END_VAR
VAR_OUTPUT
	stDataXelectrix					: ST_Xelectrix_Powerbox_OutData;				//Shows the specific output data from the Xelectric device
	stDataBatt						: ST_Battery_Output;							//{#lynus.ag#()} //Output structure with Data from Battery
	stDataBattInverter				: ST_BatteryInverter_Output;					//{#lynus.ag#()} //Output structure with Data from Battery Inverter
	stDataEMPower_Grid				: ST_ElectricMeter_Output_Power;				//Output structure with Data from Electric Meter Grid (Power Data)
	stDataEMCounter_Grid			: ST_ElectricMeter_Output_Counter;				//Output structure with Data from Electric Meter Grid (Counter Data)
	diNrOfBatt_OUT					: DINT;											//Active Number from the Battery Function for using on other functions
	diNrOfBattInverter_OUT			: DINT;											//Active Number from the Battery Inverter Function for using on other functions
	diNrOfEM_OUT_Grid				: DINT;											//Active Number from the Electric Meter for using on other functions
	lrMaxCapacityBattery_OUT		: LREAL;										//Max kWh from the Battery system. The Xelectrix System deliver this value.
	iSetpointPower_Info				: INT;											// Battery Setpoint, for monitoring purpose
END_VAR
VAR

	fbBattery						: FB_Battery;									//Function block for battery

	fbBatteryInverter				: FB_BatteryInverter;							//Function block for battery inveter

	fbEMGrid						: FB_ElectricMeter;								//Electric Meter Function 

	fbPIDChrgStandby				: FB_PID;										//Controller to control the battery current on 0 in the standby mode	

	fbNumberDeviceBattery			: FB_NumberOfDevice;							//Function block to calcualte the number of the Device

	fbNumberDeviceBatteryInvert		: FB_NumberOfDevice;							//Function block to calcualte the number of the Device

	fbNumberDeviceGrid				: FB_NumberOfDevice;							//Function block to calcualte the number of the Device

	fbMBRead_FC3					: FB_MBReadRegs;								//Modbus Read Function (FC3)

	fbMBWrite_FC16					: FB_MBWriteRegs;								//Modbus Write Function (FC16)

	fbConvertData					: FB_CV_WORD_TO_DWORD;							//Convert 2 Words in a Dword

	timDelay						: TON;											//Timer for Delay between Requests

	timTimeout						: TON;											//Timer for Timeout

	timDissableFunctions			: TON;											//Timer to dissable the Function after Lynus_Standards.Constants_General.tTimeDissableLynusFunctions Days without connection to the Lynus Cloud

	timResetConnectionOnGVL			: TON;											//Timer to try reset the connection Flag on the GVL. (When somebody delete the Connection Function and make only a onlinechange)

	timReset						: TON;											//Timer to reset the Inverter after a Error

	timErrorMTCP					: TON;											//Delay when Error on Modbus TCP

	timSetStandbyCntrl				: TOF;											//Timer to set the Standby Controller

	FPEnable						: R_TRIG;										//Internal positive Edge

	FPError_FC_3					: R_TRIG;										//Internal positive Edge

	FPError_FC_16					: R_TRIG;										//Internal positive Edge

	FPActivateControl				: R_TRIG;										//Internal positive Edge

	FNTimDissable					: F_TRIG;										//Internal negative Edge

	PD_String						: FB_PersistentData_String;						//Function to save persistent data

	arrPD							: ARRAY[1..7] OF FB_PersistentData_Number;		//Function to save persistent data

	arrBuffer_FC3					: ARRAY[1..48] OF WORD;							//Buffer with Data from FC3

	arrBuffer_FC16					: ARRAY[1..2] OF WORD;							//Buffer with Data from FC16

	arrCounterForGVL				: ARRAY[1..3] OF DINT;							//Counter to clean old data on GVL

	bEnergyGridConsReceived			: BOOL;											//Energy Consumption from Grid first time received

	bEnergyGridProdReceived			: BOOL;											//Energy Production from Grid first time received

	byWaitInStep					: BYTE;											//Wait in Step before start to clean data on PLC

	byLPWorkAroundACDevice			: BYTE;											//Loop for Workaround

	byNumberOfZero					: BYTE;											//Number with 0 Value from AC Messurement

	iSetpointPower					: INT;											//Power Setpoint in W

	iStateGVLData					: INT;											//State machine to handle the data on the GVL

	iStateModbusRead				: INT;											//State variable for Statemachine

	iStateModbusWrite				: INT;											//State variable for Statemachine

	iStateModbusError				: INT;											//State variable for Statemachine

	iStateModbus_CP					: INT;											//Compare State variable

	iMaxDcDischargeCurrentBattery	: INT;											//Variable to convert from negative to positive value

	diLPForGVL						: DINT;											//Loop to clean old data on GVL

	lrEnergyGridConsumption_CP		: LREAL;										//Energy Consumption from Grid for calculation for Workaround why Xelectrix send sometimes big value 

	lrEnergyGridProduction_CP		: LREAL;										//Energy Production from Grid for calculation for Workaround why Xelectrix send sometimes big value 
END_VAR
VAR PERSISTENT
	{attribute 'conditionalshow'}
	diNrOfEMS_IN_CP					: DINT;											//Number of EMS what control this Device to compare with the original
END_VAR

//Creator : Stefan Lackner (based on Kai Ebensperger V1)
//Company : EfficientIO
//Date : 15.12.2022
//Version : 2.0.0.0

//With this function its possible to read out values from the Xelectrix Powerbox from the factory Xelectrix
//Its also possible to controll the power in and out from Battery if its necessary.
//The protocol to the Inverter/powerbox is Modbus TCP
//When this Function is not enabled, then the Inverter is not off. But no power flows into or out of the battery.
//This Inverter deliver also the Grid power (smart Meter).
//Versions that are supported : 106
//NOTE : This Function block not support the complete emergency power mode. He switch not off when the byMaxDepthOfDischargeEPO is reached because this make the inverter by himself.

//NOTE for diNr.....Designation => 
//_IN = Here Data come in from other Functions or go out to other functions about the GVL
//_OUT = Here Data go out to other functions about the GVL

(*------------------------------------------------------------------------------------------General Input Part---------------------------------------------------------------------------------------------*)

//Check limitation
diNrOfEMS_IN := LIMIT(0,diNrOfEMS_IN,Constants_Energy.diMaxNumberOfEMS);
	
(*-------------------------------------------------------------Calcualte the number of Battery system---------------------------------------------------------------*)

fbNumberDeviceBattery(
	diActualNumberOfDevices:= Lynus_Standards.GVL_Energy.stNumberOfDevices.diNumberOfBatterys, 
	diMaxNumberOfDevices:= Constants_Energy.diMaxNumberOfBatterys, 
	udiCounterOnlineChange:= TwinCAT_SystemInfoVarList._AppInfo.OnlineChangeCnt, 
	bNumberIsCalculatet=> , 
	bFPNumberIsCalculatet=> , 
	bOnlineChange=> , 
	diNumberForThisDevice=> diNrOfBatt_OUT, 
	diNumberOfTotalDevices=> );

//Write new Numer on GVL
IF fbNumberDeviceBattery.bFPNumberIsCalculatet THEN
	Lynus_Standards.GVL_Energy.stNumberOfDevices.diNumberOfBatterys := fbNumberDeviceBattery.diNumberOfTotalDevices;	
END_IF

//Delete old Number on GVL
IF fbNumberDeviceBattery.bOnlineChange THEN 
	Lynus_Standards.GVL_Energy.stNumberOfDevices.diNumberOfBatterys := diNrOfBatt_OUT;	
		iStateGVLData := 1; 
END_IF

fbNumberDeviceBatteryInvert(
	diActualNumberOfDevices:= Lynus_Standards.GVL_Energy.stNumberOfDevices.diNumberOfBatteryInverters, 
	diMaxNumberOfDevices:= Constants_Energy.diMaxNumberOfBatteryInverters, 
	udiCounterOnlineChange:= TwinCAT_SystemInfoVarList._AppInfo.OnlineChangeCnt, 
	bNumberIsCalculatet=> , 
	bFPNumberIsCalculatet=> , 
	bOnlineChange=> , 
	diNumberForThisDevice=> diNrOfBattInverter_OUT, 
	diNumberOfTotalDevices=> );

//Write new Numer on GVL
IF fbNumberDeviceBatteryInvert.bFPNumberIsCalculatet THEN
	Lynus_Standards.GVL_Energy.stNumberOfDevices.diNumberOfBatteryInverters := fbNumberDeviceBatteryInvert.diNumberOfTotalDevices;	
END_IF

//Delete old Number on GVL
IF fbNumberDeviceBatteryInvert.bOnlineChange THEN 
	Lynus_Standards.GVL_Energy.stNumberOfDevices.diNumberOfBatteryInverters := diNrOfBattInverter_OUT;	
		iStateGVLData := 1; 
END_IF

fbNumberDeviceGrid(
	diActualNumberOfDevices:= Lynus_Standards.GVL_Energy.stNumberOfDevices.diNumberOfElectricMeters, 
	diMaxNumberOfDevices:= Constants_Energy.diMaxNumberOfElectricMeters, 
	udiCounterOnlineChange:= TwinCAT_SystemInfoVarList._AppInfo.OnlineChangeCnt, 
	bNumberIsCalculatet=> , 
	bFPNumberIsCalculatet=> , 
	bOnlineChange=> , 
	diNumberForThisDevice=> diNrOfEM_OUT_Grid, 
	diNumberOfTotalDevices=> );

//Write new Numer on GVL
IF fbNumberDeviceGrid.bFPNumberIsCalculatet THEN
	Lynus_Standards.GVL_Energy.stNumberOfDevices.diNumberOfElectricMeters := fbNumberDeviceGrid.diNumberOfTotalDevices;	
END_IF			

(*-------------------------------------------------------------Service from Backend is ready and check the connection to backend for dissabel/enable Function---------------------------------------------------------------*)

//Try to reset the variable for connection on the GVL. When all is normal then the Lynus Mqtt connection function set this variable to true in the next cycle
//When we have no connection to the backend then after Lynus_Standards.Constants_General.tTimeDissableLynusFunctions days the Function is dissabled with all of his functionalities
timResetConnectionOnGVL(IN:= NOT timResetConnectionOnGVL.Q, PT:= T#1H, Q=> , ET=> );
	IF timResetConnectionOnGVL.Q THEN Lynus_Standards.GVL_Communicator.bStateConnectionToEnableFunctions := FALSE; END_IF
		IF NOT Lynus_Standards.GVL_Communicator.bStateConnectionToEnableFunctions THEN timDissableFunctions.IN := TRUE; ELSE timDissableFunctions.IN := FALSE; END_IF  
			timDissableFunctions(IN:= , PT:= Lynus_Standards.Constants_General.tTimeDissableLynusFunctions, Q=> , ET=> );
			
(*------------------------------------------------------------------------------------------State Machine Read---------------------------------------------------------------------------------------------*)

//When the function is not enabled then the fronius control by himself without modbus tcp connection
IF NOT bEnable OR timDissableFunctions.Q THEN bActivateControl := FALSE; END_IF

// limit manual setpoint +/- 320 kW
i_SetpointPower_Manual_kW:=LIMIT(-320,i_SetpointPower_Manual_kW,320);

//Start the Statemachine
FPEnable(CLK:= bEnable, Q=> );
	FPActivateControl(CLK:= bActivateControl, Q=> );
		FNTimDissable(CLK:= timDissableFunctions.Q, Q=> );
			IF (FPEnable.Q AND iStateModbusRead = 0 AND iStateModbusRead = 0 AND iStateModbusError = 0) OR
				(bEnable AND FPActivateControl.Q AND iStateModbusRead = 0 AND iStateModbusRead = 0 AND iStateModbusError = 0) OR
					(bEnable AND FNTimDissable.Q AND iStateModbusRead = 0 AND iStateModbusRead = 0 AND iStateModbusError = 0) THEN 
						iStateModbusRead := 1; 
			END_IF
				IF NOT bEnable OR NOT bActivateControl THEN iStateModbusRead := 0; iStateModbusWrite := 0; iStateModbusError := 0; END_IF

//Timer for delay
timDelay(IN:= , PT:= T#500MS, Q=> , ET=> );

//Timer for Timeout in Statemachine
IF (iStateModbusRead > 0 AND iStateModbusRead <= 2 AND iStateModbusRead = iStateModbus_CP) OR
		(iStateModbusWrite > 0 AND iStateModbusWrite <= 1 AND iStateModbusWrite = iStateModbus_CP) THEN
			timTimeout.IN := TRUE;
ELSE	
			timTimeout.IN := FALSE;
END_IF 
	IF iStateModbusRead = 0 AND iStateModbusWrite = 0 THEN timTimeout.IN := FALSE; END_IF
		timTimeout(IN:= , PT:= T#20S, Q=> , ET=> );

CASE iStateModbusRead OF
	
	0://Init State
		iStateModbus_CP := 0;
			timDelay.IN := FALSE;
			
		stDataXelectrix.eBatteryState := E_Xelectrix_BatteryState.eNoDataReceived;
			stDataXelectrix.eGridState := E_Xelectrix_GridState.eNoDataReceived;
				stDataXelectrix.eOperatingState := E_Xelectrix_OperatingState.eNoDataReceived;	
					stDataXelectrix.bFunctionIsActive := FALSE;
			
		fbMBRead_FC3.bExecute := FALSE;
			fbMBWrite_FC16.bExecute := FALSE;	

	1://Read all the Data
		stDataXelectrix.bFunctionIsActive := TRUE;
			iStateModbus_CP := iStateModbusRead;
		
		//Reset Write
		fbMBWrite_FC16.bExecute := FALSE;
			arrBuffer_FC16[1] := 0; arrBuffer_FC16[2] := 0;
		
		//Start Read
		fbMBRead_FC3.nQuantity := 48;
			fbMBRead_FC3.nMBAddr := 0;
				fbMBRead_FC3.bExecute := TRUE;
			
		IF fbMBRead_FC3.bBusy THEN timDelay.IN := TRUE; END_IF
		
		//Wait for Delay, copy Data and then next step
		IF NOT fbMBRead_FC3.bBusy AND NOT fbMBRead_FC3.bError AND timDelay.Q THEN
			//Grid State
			IF arrBuffer_FC3[1] = 0 THEN stDataXelectrix.eGridState := E_Xelectrix_GridState.eOff; 
			ELSIF arrBuffer_FC3[1] = 1 THEN stDataXelectrix.eGridState := E_Xelectrix_GridState.eIslandMode;
			ELSIF arrBuffer_FC3[1] = 2 THEN stDataXelectrix.eGridState := E_Xelectrix_GridState.eOnline;
			ELSIF arrBuffer_FC3[1] = 3 THEN stDataXelectrix.eGridState := E_Xelectrix_GridState.eError;   	
			END_IF
			
			(*------------------------------------------Workaround why AC device deliver sometimes 0 Value--------------------------------------------------------*)
			byNumberOfZero := 0;
				FOR byLPWorkAroundACDevice := 6 TO 9 BY 1 DO
					IF arrBuffer_FC3[byLPWorkAroundACDevice] = 0 THEN byNumberOfZero := byNumberOfZero + 1; END_IF  
				END_FOR

			IF byNumberOfZero = 0 THEN
				//Real Power (Scale factor is * 100 for W)
				fbEMGrid.lrPowerTotal := INT_TO_LREAL(WORD_TO_INT(arrBuffer_FC3[2])) * 100;
				//Reactive Power (Scale factor is * 100 for var)
				fbEMGrid.lrReactivePowerTotal := INT_TO_LREAL(WORD_TO_INT(arrBuffer_FC3[3])) * 100; 
				//Frequency (Scale factor is / 100 for Hz)
				fbEMGrid.lrFrequency := INT_TO_LREAL(WORD_TO_INT(arrBuffer_FC3[6])) / 100;
				//Voltage L1/N (Scale factor is / 10 for V)
				fbEMGrid.lrVoltageL1N := INT_TO_LREAL(WORD_TO_INT(arrBuffer_FC3[7])) / 10;
				//Voltage L2/N (Scale factor is / 10 for V)
				fbEMGrid.lrVoltageL2N := INT_TO_LREAL(WORD_TO_INT(arrBuffer_FC3[8])) / 10;
				//Voltage L3/N (Scale factor is / 10 for V)
				fbEMGrid.lrVoltageL3N := INT_TO_LREAL(WORD_TO_INT(arrBuffer_FC3[9])) / 10;
				//Current L1 (Scale factor is * 100 for mA)
				fbEMGrid.lrCurrentL1 := INT_TO_LREAL(WORD_TO_INT(arrBuffer_FC3[10])) * 100;
					//Make / 1000 for A
					fbEMGrid.lrCurrentL1 := fbEMGrid.lrCurrentL1 / 1000;
				//Current L2 (Scale factor is * 100 for mA)
				fbEMGrid.lrCurrentL2 := INT_TO_LREAL(WORD_TO_INT(arrBuffer_FC3[11])) * 100;
					//Make / 1000 for A
					fbEMGrid.lrCurrentL2 := fbEMGrid.lrCurrentL2 / 1000;
				//Current L3 (Scale factor is * 100 for mA)
				fbEMGrid.lrCurrentL3 := INT_TO_LREAL(WORD_TO_INT(arrBuffer_FC3[12])) * 100;
					//Make / 1000 for A
					fbEMGrid.lrCurrentL3 := fbEMGrid.lrCurrentL3 / 1000;
			END_IF	
			(*-----------------------------------------------------------------------------------------------------------------------------------------------------*)
			
			//Max Charge Power (Scale factor is * 100 for W)
			fbBatteryInverter.rMaxChargePowerBattInverter := INT_TO_REAL(WORD_TO_INT(arrBuffer_FC3[14])) * 100; 
			//Max Discharge Power (Scale factor is * 100 for W)
			fbBatteryInverter.rMaxDischargePowerBattInverter := INT_TO_REAL(WORD_TO_INT(arrBuffer_FC3[15])) * 100;  
			
			
			r_MaxChargePower_W := LIMIT (0,r_MaxChargePower_W,fbBatteryInverter.rMaxChargePowerBattInverter);
			r_MaxDischargePower_W := LIMIT (0,r_MaxDischargePower_W,fbBatteryInverter.rMaxDischargePowerBattInverter);
			
			IF m_ManualChargeDischargeMax THEN
				fbBatteryInverter.rMaxChargePowerBattInverter := r_MaxChargePower_W;
				fbBatteryInverter.rMaxDischargePowerBattInverter := r_MaxDischargePower_W;
			END_IF
				
				//SOC (No Scalefactor. Is %)	
				fbBattery.dwBatterySOC := INT_TO_DWORD(WORD_TO_INT(arrBuffer_FC3[21]));
					fbBatteryInverter.dwBatterSOC := INT_TO_DWORD(WORD_TO_INT(arrBuffer_FC3[21]));
				//Battery Temperature (Scale factor is / 100 for °C)
				fbBattery.lrBatteryTemp := INT_TO_LREAL(WORD_TO_INT(arrBuffer_FC3[23])) / 100; 
				//Battery State
				IF arrBuffer_FC3[24] = 0 THEN stDataXelectrix.eBatteryState := E_Xelectrix_BatteryState.eOff;
				ELSIF arrBuffer_FC3[24] = 1 THEN stDataXelectrix.eBatteryState := E_Xelectrix_BatteryState.eStartUp;
				ELSIF arrBuffer_FC3[24] = 2 THEN stDataXelectrix.eBatteryState := E_Xelectrix_BatteryState.eBalancing;
				ELSIF arrBuffer_FC3[24] = 3 THEN stDataXelectrix.eBatteryState := E_Xelectrix_BatteryState.eReady;
				ELSIF arrBuffer_FC3[24] = 4 THEN stDataXelectrix.eBatteryState := E_Xelectrix_BatteryState.eOperating;
				ELSIF arrBuffer_FC3[24] = 6 THEN stDataXelectrix.eBatteryState := E_Xelectrix_BatteryState.eError;
				END_IF  
				//Operating State
				IF arrBuffer_FC3[25] = 0 THEN stDataXelectrix.eOperatingState := E_Xelectrix_OperatingState.eOff;
				ELSIF arrBuffer_FC3[25] = 1 THEN stDataXelectrix.eOperatingState := E_Xelectrix_OperatingState.eDischarge;
				ELSIF arrBuffer_FC3[25] = 2 THEN stDataXelectrix.eOperatingState := E_Xelectrix_OperatingState.eCharge;
				ELSIF arrBuffer_FC3[25] = 3 THEN stDataXelectrix.eOperatingState := E_Xelectrix_OperatingState.eIdle;
				END_IF
				//Battery Capacity in Wh (Scale factor is * 100 for Wh), but make the calculation for kWh
				lrMaxCapacityBattery_OUT := arrBuffer_FC3[26] * 100;
					lrMaxCapacityBattery_OUT := lrMaxCapacityBattery_OUT / 1000;
				//Battery Current (Scale factor is * 100 for mA)
				fbBattery.lrBatteryCurrent := INT_TO_LREAL(WORD_TO_INT(arrBuffer_FC3[27])) * 100;
					//Make / 1000 for A
					fbBattery.lrBatteryCurrent := fbBattery.lrBatteryCurrent / 1000;
						//Change the sign because in view from the Battery - is discharge and + is charge. But we use vice versa	
						fbBattery.lrBatteryCurrent := fbBattery.lrBatteryCurrent * - 1; 
				//Battery Voltage 
				fbBattery.rBatteryVoltage := INT_TO_REAL(WORD_TO_INT(arrBuffer_FC3[28]));
				//Max Charge Current (Scale factor is * 100 for mA)
				fbBattery.rMaxDcChargeCurrentBattery := INT_TO_REAL(WORD_TO_INT(arrBuffer_FC3[29])) * 100; 
					//Make / 1000 for A
					fbBattery.rMaxDcChargeCurrentBattery := fbBattery.rMaxDcChargeCurrentBattery / 1000;
				//Max Discharge Current (Scale factor is * 100 for mA)
				//Its allways a negative raw value
				iMaxDcDischargeCurrentBattery := WORD_TO_INT(arrBuffer_FC3[30]);
					iMaxDcDischargeCurrentBattery := iMaxDcDischargeCurrentBattery * - 1;
						fbBattery.rMaxDcDischargeCurrentBattery := INT_TO_REAL(iMaxDcDischargeCurrentBattery) * 100; 
					//Make / 1000 for A
					fbBattery.rMaxDcDischargeCurrentBattery := fbBattery.rMaxDcDischargeCurrentBattery / 1000;
					
			(*------------------------------------------Workaround why AC device deliver sometimes 0 Value--------------------------------------------------------*)
						//Total Production (Scale factor is * 100 for Wh)
						IF byNumberOfZero = 0 THEN 
							fbConvertData(wInputValue_1:= arrBuffer_FC3[41], wInputValue_2:= arrBuffer_FC3[42], eByteOrderForConvert:= eByteOrder.eBigEndian, dwOutputValue=> );
								//Check the difference why Xelectrix send sometimes to big value
								lrEnergyGridConsumption_CP :=  DWORD_TO_LREAL((fbConvertData.dwOutputValue * 100)) / 1000 - stDataEMCounter_Grid.lrTotalCounterEnergy_Consumption; 
									IF (lrEnergyGridConsumption_CP < 15 AND fbConvertData.dwOutputValue <> 0) OR NOT bEnergyGridConsReceived THEN 
										fbEMGrid.lrCounterEnergyT1_Consumption := fbConvertData.dwOutputValue * 100;
											fbEMGrid.lrCounterEnergyT1_Consumption := fbEMGrid.lrCounterEnergyT1_Consumption / 1000;
												fbEMGrid.lrTotalCounterEnergy_Consumption := fbEMGrid.lrCounterEnergyT1_Consumption;
									END_IF
										IF DWORD_TO_LREAL((fbConvertData.dwOutputValue * 100)) / 1000 <> 0 AND NOT bEnergyGridConsReceived THEN bEnergyGridConsReceived := TRUE; END_IF 
							//Total Consumption (Scale factor is * 100 for Wh)
							fbConvertData(wInputValue_1:= arrBuffer_FC3[43], wInputValue_2:= arrBuffer_FC3[44], eByteOrderForConvert:= eByteOrder.eBigEndian, dwOutputValue=> );
								//Check the difference why Xelectrix send sometimes to big value
								 lrEnergyGridProduction_CP :=  DWORD_TO_LREAL((fbConvertData.dwOutputValue * 100)) / 1000 - stDataEMCounter_Grid.lrTotalCounterEnergy_Production;
									IF (lrEnergyGridProduction_CP < 15 AND fbConvertData.dwOutputValue <> 0) OR NOT bEnergyGridProdReceived THEN 
										fbEMGrid.lrCounterEnergyT1_Production := fbConvertData.dwOutputValue * 100;
											fbEMGrid.lrCounterEnergyT1_Production := fbEMGrid.lrCounterEnergyT1_Production / 1000;
												fbEMGrid.lrTotalCounterEnergy_Production := fbEMGrid.lrCounterEnergyT1_Production;
									END_IF
										IF DWORD_TO_LREAL((fbConvertData.dwOutputValue * 100)) / 1000 <> 0 AND NOT bEnergyGridProdReceived THEN bEnergyGridProdReceived := TRUE; END_IF 
						END_IF
			(*-----------------------------------------------------------------------------------------------------------------------------------------------------*)		
						
			//Go to Next Step
			fbMBRead_FC3.bExecute := FALSE;
				timDelay.IN := FALSE;		
					iStateModbusRead := 2;
		END_IF
		
		//Xelectrics Grid Error
		IF NOT fbMBRead_FC3.bBusy AND NOT fbMBRead_FC3.bError AND timDelay.Q AND stDataXelectrix.eGridState = E_Xelectrix_GridState.eError THEN
			iStateModbusError := 300;
				stDataXelectrix.eErrorState := E_Xelectrix_Error.eXelectrixError;
		END_IF
			//Xelectrics Battery Error
			IF NOT fbMBRead_FC3.bBusy AND NOT fbMBRead_FC3.bError AND timDelay.Q AND stDataXelectrix.eBatteryState = E_Xelectrix_BatteryState.eError THEN
				iStateModbusError := 300;
					stDataXelectrix.eErrorState := E_Xelectrix_Error.eXelectrixError;
			END_IF
		
		//Error or Timeout
		IF FPError_FC_3.Q OR timTimeout.Q THEN
			iStateModbusError := 300;
				stDataXelectrix.eErrorState := E_Xelectrix_Error.eModbusTCPError;
		END_IF
	
	2://Wait 1 Step to reset the delay counter befor start to write
		iStateModbus_CP := iStateModbusRead;
		
			iStateModbusWrite := 1;
				iStateModbusRead := - 1;	
				
		//Timeout
		IF timTimeout.Q THEN
			iStateModbusError := 300;
				stDataXelectrix.eErrorState := E_Xelectrix_Error.eModbusTCPError;
		END_IF
		
END_CASE

(*----------------------------------------------------------------------------------------Battery Inverter Function----------------------------------------------------------------------------------------------*)

//Error and Reset
timErrorMTCP(IN:= stDataXelectrix.bError AND stDataXelectrix.eErrorState = E_Xelectrix_Error.eModbusTCPError, PT:= T#5S, Q=> , ET=> );

IF timDissableFunctions.Q THEN fbBatteryInverter.bWarning := TRUE; fbBatteryInverter.iWarningCode := 0; ELSE fbBatteryInverter.bWarning := FALSE; END_IF 
	IF (stDataXelectrix.bError AND stDataXelectrix.eBatteryState = E_Xelectrix_BatteryState.eError) OR timErrorMTCP.Q OR Lynus_Standards.GVL_Energy.stNumberOfDevices.diNumberOfBatteryInverters > Constants_Energy.diMaxNumberOfBatteryInverters THEN fbBatteryInverter.bError := TRUE; ELSE fbBatteryInverter.bError := FALSE; END_IF	
		IF Lynus_Standards.GVL_Energy.stNumberOfDevices.diNumberOfBatteryInverters > Constants_Energy.diMaxNumberOfBatteryInverters THEN fbBatteryInverter.iErrorCode := 1;
		ELSIF stDataXelectrix.bError THEN fbBatteryInverter.iErrorCode := 0; 
		END_IF  

//Autoreset after Error, because Xelectrix deleiver somtimes a Error and they dont know why.....
timReset(IN:= stDataBattInverter.byErrorWarning <> 0 AND NOT timReset.Q, PT:= T#1S, Q=> , ET=> );	
		
//Island mode active
IF stDataXelectrix.eGridState = E_Xelectrix_GridState.eIslandMode THEN fbBatteryInverter.bWorkOnIslandMode := TRUE; ELSE fbBatteryInverter.bWorkOnIslandMode := FALSE; END_IF
		
//Function
fbBatteryInverter(
	bEnable:= bEnable AND NOT timDissableFunctions.Q, 
	bInverterOnOff:= TRUE, 
	bError:= , 
	bWarning:= , 
	bReset:= bReset OR timReset.Q,  
	bWorkOnIslandMode:= , 
	bWriteWithDelay:= TRUE, 
	byPriority:= byPriority, 
	byReserveSOCEPO:= Lynus_Standards.GVL_Energy.stDataOfBatteryInverters[diNrOfEMS_IN,diNrOfBattInverter_OUT].byReserveSOCEPO, 
	byMaxDepthOfDischargeEPO:= Lynus_Standards.GVL_Energy.stDataOfBatteryInverters[diNrOfEMS_IN,diNrOfBattInverter_OUT].byMaxDepthOfDischargeEPO, 
	iErrorCode:= , 
	iWarningCode:= , 
	dwBatterSOC:= , 
	rTargetPower:= Lynus_Standards.GVL_Energy.stDataOfBatteryInverters[diNrOfEMS_IN,diNrOfBattInverter_OUT].rTargetPowerEMS, 
	lrActualBatteryPower:= fbBattery.lrBatteryCurrent * fbBattery.rBatteryVoltage, 
	rMaxChargePowerBattInverter:= , 
	rMaxDischargePowerBattInverter:= , 
	lrBattInverterPowerOnIslandMode:= 0, 
	lrBattInverterPowerOnNormalMode:= 0, 
	tTimDelayOutput:= T#5S, 
	stDataBattInvertOut=> , 
	stDataBattInvertOutDelay=> stDataBattInverter);

//Controller to hold the Battery Current to 0 and take the rest from the Grid. (Avoid discharge in standby or when reaching the reserve charge for EPO)
timSetStandbyCntrl(IN:= fbBatteryInverter.stDataBattInvertOut.rTargetPower = 0, PT:= T#5S, Q=> , ET=> );

IF timSetStandbyCntrl.Q AND bEnable AND bActivateControl THEN
	fbPIDChrgStandby.bEnable := TRUE;
		//Charge the Battery when its under the reserve for SOC
		IF fbBatteryInverter.dwBatterSOC < fbBatteryInverter.byReserveSOCEPO THEN
			fbPIDChrgStandby.rSetpoint := (fbBattery.stDataBatteryOut.rMaxDcChargeCurrent * 0.1) * - 1; 	
		ELSE
			fbPIDChrgStandby.rSetpoint := 0;	
		END_IF		 
ELSE
	fbPIDChrgStandby.bEnable := FALSE;
END_IF

fbPIDChrgStandby( 
	bEnable:= , 
	rSetpoint:= , 
	udiIValue:= 750, 
	udiDValue:= 0, 
	udiDamping:= 0, 
	rPValue:= 0.32, 
	rMaxValue:= 0, 
	rMinValue:= ((fbBatteryInverter.rMaxChargePowerBattInverter / 100) * - 1) / 2, 
	rNeutralZone:= 0.1, 
	bDirection:= FALSE, 
	rActualValue:= LREAL_TO_REAL(fbBattery.stDataBatteryOut.lrCurrent), 
	rQController=> );	

//Set the Target power to a fixed value when the controller is acitve
IF fbPIDChrgStandby.bEnable THEN 
	stDataBattInverter.rTargetPower := - 1;
END_IF
	
(*----------------------------------------------------------------------------------------Battery Function----------------------------------------------------------------------------------------------*)

//Error
IF timDissableFunctions.Q THEN fbBattery.bWarning := TRUE; fbBattery.iWarningCode := 0; ELSE fbBattery.bWarning := FALSE; END_IF 
	IF (stDataXelectrix.bError AND stDataXelectrix.eBatteryState = E_Xelectrix_BatteryState.eError) OR timErrorMTCP.Q OR Lynus_Standards.GVL_Energy.stNumberOfDevices.diNumberOfBatterys > Constants_Energy.diMaxNumberOfBatterys THEN fbBattery.bError := TRUE; ELSE fbBattery.bError := FALSE; END_IF
		IF Lynus_Standards.GVL_Energy.stNumberOfDevices.diNumberOfBatterys > Constants_Energy.diMaxNumberOfBatterys THEN fbBattery.iErrorCode := 1;
		ELSIF stDataXelectrix.bError THEN fbBattery.iErrorCode := 0; 
		END_IF

//Function
fbBattery(
	bEnable:= bEnable AND NOT timDissableFunctions.Q, 
	bError:= , 
	bWarning:= , 
	bCalculatePower:= TRUE, 
	bReset:= bReset OR timReset.Q, 
	bWriteWithDelay:= TRUE, 
	iErrorCode:= , 
	iWarningCode:= , 
	dwBatterySOC:= , 
	dwBatterySOH:= 0, 
	rBatteryVoltage:= , 
	rMaxDcChargeCurrentBattery:= , 
	rMaxDcDischargeCurrentBattery:= , 
	rMaxChargeVoltage:= 0, 
	lrMaxCapacityBattery:= lrMaxCapacityBattery, 
	lrBatteryPower:= 0, 
	lrBatteryCurrent:= , 
	lrBatteryTemp:= , 
	tTimDelayOutput:= T#5S, 
	stDataBatteryOut=> , 
	stDataBatteryOutDelay=> stDataBatt);

(*----------------------------------------------------------------------------------------Electric Meter Function for Grid----------------------------------------------------------------------------------------------*)

//Error
IF timDissableFunctions.Q THEN fbEMGrid.bWarning := TRUE; fbEMGrid.iWarningCode := 0; ELSE fbEMGrid.bWarning := FALSE; END_IF 
	IF (stDataXelectrix.bError AND stDataXelectrix.eGridState = E_Xelectrix_GridState.eError) OR timErrorMTCP.Q OR Lynus_Standards.GVL_Energy.stNumberOfDevices.diNumberOfElectricMeters > Constants_Energy.diMaxNumberOfElectricMeters THEN fbEMGrid.bError := TRUE; ELSE fbEMGrid.bError := FALSE; END_IF
		IF Lynus_Standards.GVL_Energy.stNumberOfDevices.diNumberOfElectricMeters > Constants_Energy.diMaxNumberOfElectricMeters THEN fbEMGrid.iErrorCode := 1;
		ELSIF stDataXelectrix.bError THEN fbEMGrid.iErrorCode := 0;
		END_IF  

//Read Out Data done for EM Function
IF iStateModbusRead <> 1 THEN fbEMGrid.bReadOutDataDone := TRUE; ELSE fbEMGrid.bReadOutDataDone := FALSE; END_IF		
		
//Function
fbEMGrid(
	bEnable:= bEnable AND NOT timDissableFunctions.Q, 
	bError:= , 
	bEnableReadOutFunction:= FALSE, 
	bWriteWithDelay:= TRUE, 
	bPowerDataInvers:= FALSE,
	bReadOutDataDone:= ,
	iTimeReadOutInterval:= , 
	iErrorCode:= , 
	iWarningCode:= , 
	lrTotalCounterEnergy_Consumption:= , 
	lrTotalCounterEnergy_Production:= , 
	lrCounterEnergyT1_Consumption:= , 
	lrCounterEnergyT2_Consumption:= 0, 
	lrCounterEnergyT1_Production:= , 
	lrCounterEnergyT2_Production:= 0, 
	lrCurrentL1:= , 
	lrVoltageL1N:= , 
	lrVoltageL1L2:= 0, 
	lrPowerL1:= 0, 
	lrCurrentL2:= , 
	lrVoltageL2N:= , 
	lrVoltageL2L3:= 0, 
	lrPowerL2:= 0, 
	lrCurrentL3:= , 
	lrVoltageL3N:= , 
	lrVoltageL3L1:= 0, 
	lrPowerL3:= 0, 
	lrPowerTotal:= , 
	lrFrequency:= , 
	lrReactivePowerTotal:= , 
	lrApparentPowerTotal:= 0, 
	tTimDelayOutput:= T#5S, 
	stDataEMOutPower=> , 
	stDataEMOutPowerDelay=> stDataEMPower_Grid, 
	stDataEMOutCounter=> ,
	stDataEMOutCounterDelay=> stDataEMCounter_Grid,  
	bReadOutMeter=> );

(*------------------------------------------------------------------------------------------State Machine Write---------------------------------------------------------------------------------------------*)	
	
CASE iStateModbusWrite OF	
	
	1://Setpoint for Power and set the Timout on Inverter to 10 Seconds. (When after this time the inverter not received a new Message over Modbus TCP, then he goes back in his own automatic mode and work by himself)
		iStateModbus_CP := iStateModbusWrite;	
		
		fbMBWrite_FC16.nQuantity := 2;
			fbMBWrite_FC16.nMBAddr := 100;
				fbMBWrite_FC16.bExecute := TRUE;
		
		//Setpoint for the Power when discharge (Scale factor is / 100 for W on the Inverter) 
		IF fbBatteryInverter.stDataBattInvertOut.rTargetPower >= 0 THEN
			IF ((fbBatteryInverter.stDataBattInvertOut.rMaxDischargePower * 1000) * (fbBatteryInverter.stDataBattInvertOut.rTargetPower / 100)) / 100 >= - 32768 AND 
				((fbBatteryInverter.stDataBattInvertOut.rMaxDischargePower * 1000) * (fbBatteryInverter.stDataBattInvertOut.rTargetPower / 100)) / 100 <= 32767 THEN
					iSetpointPower := REAL_TO_INT(((fbBatteryInverter.stDataBattInvertOut.rMaxDischargePower * 1000) * (fbBatteryInverter.stDataBattInvertOut.rTargetPower / 100)) / 100);  
						arrBuffer_FC16[1] := INT_TO_WORD(iSetpointPower);
			END_IF
		END_IF
		//Setpoint for the Power when charge (Scale factor is / 100 for W on the Inverter) 
		IF fbBatteryInverter.stDataBattInvertOut.rTargetPower < 0 OR fbPIDChrgStandby.bEnable THEN
			IF ((fbBatteryInverter.stDataBattInvertOut.rMaxChargePower * 1000) * (fbBatteryInverter.stDataBattInvertOut.rTargetPower / 100)) / 100 >= - 32768 AND 
				((fbBatteryInverter.stDataBattInvertOut.rMaxChargePower * 1000) * (fbBatteryInverter.stDataBattInvertOut.rTargetPower / 100)) / 100 <= 32767 THEN
					iSetpointPower := REAL_TO_INT(((fbBatteryInverter.stDataBattInvertOut.rMaxChargePower * 1000) * (fbBatteryInverter.stDataBattInvertOut.rTargetPower / 100)) / 100);  
						//Take the Setpoint from the Standby Controller
						IF fbPIDChrgStandby.bEnable AND fbPIDChrgStandby.rQController <= 0 AND fbPIDChrgStandby.rQController >= -32768 THEN
							iSetpointPower := REAL_TO_INT(fbPIDChrgStandby.rQController);  
						END_IF
					arrBuffer_FC16[1] := INT_TO_WORD(iSetpointPower); 
			END_IF
		END_IF
		//manual operation setpoint, for testing pupose only!
		IF m_ManualSetpointEnable THEN
			arrBuffer_FC16[1] := INT_TO_WORD(i_SetpointPower_Manual_kW*10); 
		END_IF
		iSetpointPower_Info := WORD_TO_INT(arrBuffer_FC16[1]);
		//Timeout Time
		arrBuffer_FC16[2] := 10;
		
		IF fbMBWrite_FC16.bBusy THEN timDelay.IN := TRUE; END_IF

		//Wait for Delay and then next step
		IF NOT fbMBWrite_FC16.bBusy AND NOT fbMBWrite_FC16.bError AND timDelay.Q THEN
			fbMBWrite_FC16.bExecute := FALSE;
				timDelay.IN := FALSE;
					stDataXelectrix.bError := FALSE; 
						stDataXelectrix.eErrorState := E_Xelectrix_Error.eNoError;
							//Restart from new with the Read out part
							iStateModbusRead := 1;
								iStateModbusWrite := 0;
		END_IF
				
		//Error or Timout
		IF FPError_FC_16.Q OR timTimeout.Q THEN
			iStateModbusError := 300;
				stDataXelectrix.eErrorState := E_Xelectrix_Error.eModbusTCPError;
		END_IF

END_CASE

(*------------------------------------------------------------------------------------------State Machine Write---------------------------------------------------------------------------------------------*)	

CASE iStateModbusError OF
	
	300://Error
		iStateModbus_CP := iStateModbusError;
		timDelay.IN := FALSE;
		fbMBRead_FC3.bExecute := FALSE;
		fbMBWrite_FC16.bExecute := FALSE;
		stDataXelectrix.bError := TRUE;	
		//Restart from new with the Read out part after an Error
		iStateModbusRead := 1;	
		iStateModbusError := 0;
		iStateModbusWrite := 0;	
END_CASE

(*------------------------------------------------------------------------------------------Modbus TCP Functions---------------------------------------------------------------------------------------------*)

fbMBRead_FC3(	sIPAddr:= sIPAdress, 
				nUnitID := byUnitID, 
				nTCPPort:= 502, 
				cbLength:= SIZEOF(arrBuffer_FC3), 
				pDestAddr:= ADR(arrBuffer_FC3), 
				tTimeout:= T#10S );
FPError_FC_3(CLK:= fbMBRead_FC3.bError, Q=> );

fbMBWrite_FC16(	sIPAddr:= sIPAdress, 
				nTCPPort:= 502, 
				nUnitID := byUnitID, 
				cbLength:= SIZEOF(arrBuffer_FC16), 
				pSrcAddr:= ADR(arrBuffer_FC16), 
				tTimeout:= T#10S );
				
FPError_FC_16(CLK:= fbMBWrite_FC16.bError, Q=> );

(*-----------------------------------------------------------Handle data to Global structure for al Devices that are included in this function-----------------------------------------------------------------*)

//Delete al old Data on GVL after a online change or change on the variable diNrOfEMS_IDOD
IF diNrOfEMS_IN <> diNrOfEMS_IN_CP AND iStateGVLData = 0 THEN iStateGVLData := 10; END_IF 

CASE iStateGVLData OF
	
	0://Init Step
		byWaitInStep := 0;
			arrCounterForGVL[1] := 1; arrCounterForGVL[2] := 1; arrCounterForGVL[3] := 1;
	
	1://Wait for 4 Steps before clean al Data on GVL
		byWaitInStep := byWaitInStep + 1;
			IF (byWaitInStep >= 4 AND (fbNumberDeviceBattery.bNumberIsCalculatet OR fbNumberDeviceBatteryInvert.bNumberIsCalculatet OR fbNumberDeviceGrid.bNumberIsCalculatet)) THEN iStateGVLData := 2; END_IF
				//To much Devices, back to the Init step
				IF byWaitInStep >= 4 AND NOT fbNumberDeviceBattery.bNumberIsCalculatet AND NOT fbNumberDeviceBatteryInvert.bNumberIsCalculatet AND NOT fbNumberDeviceGrid.bNumberIsCalculatet THEN iStateGVLData := 0; END_IF	
			
	2://Clear all Data in GVL
		FOR diLPForGVL := 1 TO Constants_Energy.diMaxNumberOfEMS BY 1 DO
			//Battery Inverters 
			IF fbNumberDeviceBatteryInvert.bNumberIsCalculatet THEN 
				Lynus_Standards.GVL_Energy.stDataOfBatteryInverters[diLPForGVL,arrCounterForGVL[1]].bEnabled := FALSE;
					Lynus_Standards.GVL_Energy.stDataOfBatteryInverters[diLPForGVL,arrCounterForGVL[1]].bOnOff := FALSE;
						Lynus_Standards.GVL_Energy.stDataOfBatteryInverters[diLPForGVL,arrCounterForGVL[1]].bWorkOnIslandMode := FALSE;
							Lynus_Standards.GVL_Energy.stDataOfBatteryInverters[diLPForGVL,arrCounterForGVL[1]].byErrorWarning := 0;
								Lynus_Standards.GVL_Energy.stDataOfBatteryInverters[diLPForGVL,arrCounterForGVL[1]].byPriority := 0;
									Lynus_Standards.GVL_Energy.stDataOfBatteryInverters[diLPForGVL,arrCounterForGVL[1]].dwBatterySOC := 0;
										Lynus_Standards.GVL_Energy.stDataOfBatteryInverters[diLPForGVL,arrCounterForGVL[1]].lrPowerOnIslandMode := 0;
											Lynus_Standards.GVL_Energy.stDataOfBatteryInverters[diLPForGVL,arrCounterForGVL[1]].rMaxChargePower := 0;
												Lynus_Standards.GVL_Energy.stDataOfBatteryInverters[diLPForGVL,arrCounterForGVL[1]].rMaxDischargePower := 0;
													Lynus_Standards.GVL_Energy.stDataOfBatteryInverters[diLPForGVL,arrCounterForGVL[1]].lrPowerNormalMode := 0;
														//Set also the target value from ems back here to 0 and not in EMS function because EMS is in Standy when we have a online change (Problem when we delete a ems function and make a online change)
														Lynus_Standards.GVL_Energy.stDataOfBatteryInverters[diLPForGVL,arrCounterForGVL[1]].rTargetPowerEMS := 0;
															Lynus_Standards.GVL_Energy.stDataOfBatteryInverters[diLPForGVL,arrCounterForGVL[1]].byMaxDepthOfDischargeEPO := 0;
																Lynus_Standards.GVL_Energy.stDataOfBatteryInverters[diLPForGVL,arrCounterForGVL[1]].byReserveSOCEPO := 0;
			END_IF
				//Batterys 
				IF fbNumberDeviceBattery.bNumberIsCalculatet THEN 
					Lynus_Standards.GVL_Energy.stDataOfBatterys[diLPForGVL,arrCounterForGVL[2]].bEnabled := FALSE;
						Lynus_Standards.GVL_Energy.stDataOfBatterys[diLPForGVL,arrCounterForGVL[2]].byErrorWarning := 0;
							Lynus_Standards.GVL_Energy.stDataOfBatterys[diLPForGVL,arrCounterForGVL[2]].dwSOC := 0;
								Lynus_Standards.GVL_Energy.stDataOfBatterys[diLPForGVL,arrCounterForGVL[2]].dwSOH := 0;
									Lynus_Standards.GVL_Energy.stDataOfBatterys[diLPForGVL,arrCounterForGVL[2]].lrCapacity := 0;
										Lynus_Standards.GVL_Energy.stDataOfBatterys[diLPForGVL,arrCounterForGVL[2]].lrCurrent := 0;
											Lynus_Standards.GVL_Energy.stDataOfBatterys[diLPForGVL,arrCounterForGVL[2]].lrPower := 0;
												Lynus_Standards.GVL_Energy.stDataOfBatterys[diLPForGVL,arrCounterForGVL[2]].lrPowerConsumption := 0;
													Lynus_Standards.GVL_Energy.stDataOfBatterys[diLPForGVL,arrCounterForGVL[2]].lrPowerProduction := 0;
														Lynus_Standards.GVL_Energy.stDataOfBatterys[diLPForGVL,arrCounterForGVL[2]].lrTemp := 0;
															Lynus_Standards.GVL_Energy.stDataOfBatterys[diLPForGVL,arrCounterForGVL[2]].rMaxChargeVoltage := 0;
																Lynus_Standards.GVL_Energy.stDataOfBatterys[diLPForGVL,arrCounterForGVL[2]].rMaxDcChargeCurrent := 0;
																	Lynus_Standards.GVL_Energy.stDataOfBatterys[diLPForGVL,arrCounterForGVL[2]].rMaxDcDischargeCurrent := 0;
																		Lynus_Standards.GVL_Energy.stDataOfBatterys[diLPForGVL,arrCounterForGVL[2]].rVoltage := 0;
				END_IF
		END_FOR
			//Electric Meter Grid
			IF fbNumberDeviceGrid.bNumberIsCalculatet THEN 
				Lynus_Standards.GVL_Energy.stDataElectricMeters[arrCounterForGVL[3]].bEnabled := FALSE;	
					Lynus_Standards.GVL_Energy.stDataElectricMeters[arrCounterForGVL[3]].byErrorWarning := 0;
						Lynus_Standards.GVL_Energy.stDataElectricMeters[arrCounterForGVL[3]].lrCounterEnergyT1_Consumption := 0;
							Lynus_Standards.GVL_Energy.stDataElectricMeters[arrCounterForGVL[3]].lrCounterEnergyT1_Production := 0;
								Lynus_Standards.GVL_Energy.stDataElectricMeters[arrCounterForGVL[3]].lrCounterEnergyT2_Consumption := 0;
									Lynus_Standards.GVL_Energy.stDataElectricMeters[arrCounterForGVL[3]].lrCounterEnergyT2_Production := 0;
										Lynus_Standards.GVL_Energy.stDataElectricMeters[arrCounterForGVL[3]].lrPower := 0;
											Lynus_Standards.GVL_Energy.stDataElectricMeters[arrCounterForGVL[3]].lrPowerConsumption := 0;
												Lynus_Standards.GVL_Energy.stDataElectricMeters[arrCounterForGVL[3]].lrPowerProduction := 0;
													Lynus_Standards.GVL_Energy.stDataElectricMeters[arrCounterForGVL[3]].lrTotalCounterEnergy_Consumption := 0;
														Lynus_Standards.GVL_Energy.stDataElectricMeters[arrCounterForGVL[3]].lrTotalCounterEnergy_Production := 0;
			END_IF
		
			//Counter for Battery Inverter
			arrCounterForGVL[1] := arrCounterForGVL[1] + 1;
				arrCounterForGVL[1] := LIMIT(0,arrCounterForGVL[1],Constants_Energy.diMaxNumberOfBatteryInverters);
			//Counter for Batterys
			arrCounterForGVL[2] := arrCounterForGVL[2] + 1;
				arrCounterForGVL[2] := LIMIT(0,arrCounterForGVL[2],Constants_Energy.diMaxNumberOfBatterys);
			//Electric Meters
			arrCounterForGVL[3] := arrCounterForGVL[3] + 1;
				arrCounterForGVL[3] := LIMIT(0,arrCounterForGVL[3],Constants_Energy.diMaxNumberOfElectricMeters);
					//Back to the init step
					IF arrCounterForGVL[1] >= Constants_Energy.diMaxNumberOfBatteryInverters AND arrCounterForGVL[2] >= Constants_Energy.diMaxNumberOfBatterys AND  
						arrCounterForGVL[3] >= Constants_Energy.diMaxNumberOfElectricMeters THEN 
							iStateGVLData := 0; 
					END_IF

	10://Clear old Data on GVL 		
		//Battery Inverter
		Lynus_Standards.GVL_Energy.stDataOfBatteryInverters[diNrOfEMS_IN_CP,diNrOfBattInverter_OUT].bEnabled := FALSE;
			Lynus_Standards.GVL_Energy.stDataOfBatteryInverters[diNrOfEMS_IN_CP,diNrOfBattInverter_OUT].bOnOff := FALSE;
				Lynus_Standards.GVL_Energy.stDataOfBatteryInverters[diNrOfEMS_IN_CP,diNrOfBattInverter_OUT].bWorkOnIslandMode := FALSE;
					Lynus_Standards.GVL_Energy.stDataOfBatteryInverters[diNrOfEMS_IN_CP,diNrOfBattInverter_OUT].byErrorWarning := 0;
						Lynus_Standards.GVL_Energy.stDataOfBatteryInverters[diNrOfEMS_IN_CP,diNrOfBattInverter_OUT].byPriority := 0;
							Lynus_Standards.GVL_Energy.stDataOfBatteryInverters[diNrOfEMS_IN_CP,diNrOfBattInverter_OUT].dwBatterySOC := 0;
								Lynus_Standards.GVL_Energy.stDataOfBatteryInverters[diNrOfEMS_IN_CP,diNrOfBattInverter_OUT].lrPowerOnIslandMode := 0;
									Lynus_Standards.GVL_Energy.stDataOfBatteryInverters[diNrOfEMS_IN_CP,diNrOfBattInverter_OUT].rMaxChargePower := 0;
										Lynus_Standards.GVL_Energy.stDataOfBatteryInverters[diNrOfEMS_IN_CP,diNrOfBattInverter_OUT].rMaxDischargePower := 0;
											Lynus_Standards.GVL_Energy.stDataOfBatteryInverters[diNrOfEMS_IN_CP,diNrOfBattInverter_OUT].lrPowerNormalMode := 0;
		//Batterys		
		Lynus_Standards.GVL_Energy.stDataOfBatterys[diNrOfEMS_IN_CP,diNrOfBatt_OUT].bEnabled := FALSE;
			Lynus_Standards.GVL_Energy.stDataOfBatterys[diNrOfEMS_IN_CP,diNrOfBatt_OUT].byErrorWarning := 0;
				Lynus_Standards.GVL_Energy.stDataOfBatterys[diNrOfEMS_IN_CP,diNrOfBatt_OUT].dwSOC := 0;
					Lynus_Standards.GVL_Energy.stDataOfBatterys[diNrOfEMS_IN_CP,diNrOfBatt_OUT].dwSOH := 0;
						Lynus_Standards.GVL_Energy.stDataOfBatterys[diNrOfEMS_IN_CP,diNrOfBatt_OUT].lrCapacity := 0;
							Lynus_Standards.GVL_Energy.stDataOfBatterys[diNrOfEMS_IN_CP,diNrOfBatt_OUT].lrCurrent := 0;
								Lynus_Standards.GVL_Energy.stDataOfBatterys[diNrOfEMS_IN_CP,diNrOfBatt_OUT].lrPower := 0;
									Lynus_Standards.GVL_Energy.stDataOfBatterys[diNrOfEMS_IN_CP,diNrOfBatt_OUT].lrPowerConsumption := 0;
										Lynus_Standards.GVL_Energy.stDataOfBatterys[diNrOfEMS_IN_CP,diNrOfBatt_OUT].lrPowerProduction := 0;
											Lynus_Standards.GVL_Energy.stDataOfBatterys[diNrOfEMS_IN_CP,diNrOfBatt_OUT].lrTemp := 0;
												Lynus_Standards.GVL_Energy.stDataOfBatterys[diNrOfEMS_IN_CP,diNrOfBatt_OUT].rMaxChargeVoltage := 0;
													Lynus_Standards.GVL_Energy.stDataOfBatterys[diNrOfEMS_IN_CP,diNrOfBatt_OUT].rMaxDcChargeCurrent := 0;
														Lynus_Standards.GVL_Energy.stDataOfBatterys[diNrOfEMS_IN_CP,diNrOfBatt_OUT].rMaxDcDischargeCurrent := 0;
															Lynus_Standards.GVL_Energy.stDataOfBatterys[diNrOfEMS_IN_CP,diNrOfBatt_OUT].rVoltage := 0;
									
		diNrOfEMS_IN_CP := diNrOfEMS_IN;
			//Back to the init step
			iStateGVLData := 0;

END_CASE 	 

//Write Data on GVL for Battery Inverter
IF diNrOfBattInverter_OUT > 0 AND fbNumberDeviceBatteryInvert.bNumberIsCalculatet AND diNrOfEMS_IN > 0 THEN
	Lynus_Standards.GVL_Energy.stDataOfBatteryInverters[diNrOfEMS_IN,diNrOfBattInverter_OUT].bEnabled := fbBatteryInverter.stDataBattInvertOut.bEnabled;
		Lynus_Standards.GVL_Energy.stDataOfBatteryInverters[diNrOfEMS_IN,diNrOfBattInverter_OUT].bOnOff := fbBatteryInverter.stDataBattInvertOut.bOnOff;
			Lynus_Standards.GVL_Energy.stDataOfBatteryInverters[diNrOfEMS_IN,diNrOfBattInverter_OUT].bWorkOnIslandMode := fbBatteryInverter.stDataBattInvertOut.bWorkOnIslandMode;
				Lynus_Standards.GVL_Energy.stDataOfBatteryInverters[diNrOfEMS_IN,diNrOfBattInverter_OUT].byErrorWarning := fbBatteryInverter.stDataBattInvertOut.byErrorWarning;
					Lynus_Standards.GVL_Energy.stDataOfBatteryInverters[diNrOfEMS_IN,diNrOfBattInverter_OUT].byPriority := fbBatteryInverter.stDataBattInvertOut.byPriority;
						Lynus_Standards.GVL_Energy.stDataOfBatteryInverters[diNrOfEMS_IN,diNrOfBattInverter_OUT].dwBatterySOC := fbBatteryInverter.dwBatterSOC;
							Lynus_Standards.GVL_Energy.stDataOfBatteryInverters[diNrOfEMS_IN,diNrOfBattInverter_OUT].lrPowerOnIslandMode := fbBatteryInverter.stDataBattInvertOut.lrPowerOnIslandMode;	
								Lynus_Standards.GVL_Energy.stDataOfBatteryInverters[diNrOfEMS_IN,diNrOfBattInverter_OUT].rMaxChargePower := fbBatteryInverter.stDataBattInvertOut.rMaxChargePower;
									Lynus_Standards.GVL_Energy.stDataOfBatteryInverters[diNrOfEMS_IN,diNrOfBattInverter_OUT].rMaxDischargePower := fbBatteryInverter.stDataBattInvertOut.rMaxDischargePower;
										Lynus_Standards.GVL_Energy.stDataOfBatteryInverters[diNrOfEMS_IN,diNrOfBattInverter_OUT].lrPowerNormalMode := fbBatteryInverter.stDataBattInvertOut.lrPowerNormalMode;	
END_IF 
	//Write Data on GVL for Batterys
	IF diNrOfBatt_OUT > 0 AND fbNumberDeviceBattery.bNumberIsCalculatet AND diNrOfEMS_IN > 0 THEN
		Lynus_Standards.GVL_Energy.stDataOfBatterys[diNrOfEMS_IN,diNrOfBatt_OUT].bEnabled := fbBattery.stDataBatteryOut.bEnabled;	
			Lynus_Standards.GVL_Energy.stDataOfBatterys[diNrOfEMS_IN,diNrOfBatt_OUT].byErrorWarning := fbBattery.stDataBatteryOut.byErrorWarning;
				Lynus_Standards.GVL_Energy.stDataOfBatterys[diNrOfEMS_IN,diNrOfBatt_OUT].dwSOC := fbBattery.stDataBatteryOut.dwSOC;
					Lynus_Standards.GVL_Energy.stDataOfBatterys[diNrOfEMS_IN,diNrOfBatt_OUT].dwSOH := fbBattery.stDataBatteryOut.dwSOH;
						Lynus_Standards.GVL_Energy.stDataOfBatterys[diNrOfEMS_IN,diNrOfBatt_OUT].lrCapacity := fbBattery.stDataBatteryOut.lrCapacity;
							Lynus_Standards.GVL_Energy.stDataOfBatterys[diNrOfEMS_IN,diNrOfBatt_OUT].lrCurrent := fbBattery.stDataBatteryOut.lrCurrent;
								Lynus_Standards.GVL_Energy.stDataOfBatterys[diNrOfEMS_IN,diNrOfBatt_OUT].lrPower := fbBattery.stDataBatteryOut.lrPower;
									Lynus_Standards.GVL_Energy.stDataOfBatterys[diNrOfEMS_IN,diNrOfBatt_OUT].lrPowerConsumption := fbBattery.stDataBatteryOut.lrPowerConsumption;
										Lynus_Standards.GVL_Energy.stDataOfBatterys[diNrOfEMS_IN,diNrOfBatt_OUT].lrPowerProduction := fbBattery.stDataBatteryOut.lrPowerProduction;
											Lynus_Standards.GVL_Energy.stDataOfBatterys[diNrOfEMS_IN,diNrOfBatt_OUT].lrTemp := fbBattery.stDataBatteryOut.lrTemp;
												Lynus_Standards.GVL_Energy.stDataOfBatterys[diNrOfEMS_IN,diNrOfBatt_OUT].rMaxChargeVoltage := fbBattery.stDataBatteryOut.rMaxChargeVoltage;
													Lynus_Standards.GVL_Energy.stDataOfBatterys[diNrOfEMS_IN,diNrOfBatt_OUT].rMaxDcChargeCurrent := fbBattery.stDataBatteryOut.rMaxDcChargeCurrent;
														Lynus_Standards.GVL_Energy.stDataOfBatterys[diNrOfEMS_IN,diNrOfBatt_OUT].rMaxDcDischargeCurrent := fbBattery.stDataBatteryOut.rMaxDcDischargeCurrent;
															Lynus_Standards.GVL_Energy.stDataOfBatterys[diNrOfEMS_IN,diNrOfBatt_OUT].rVoltage := fbBattery.stDataBatteryOut.rBatteryVoltage;
	END_IF
//Write Data on GVL for Electric Meter (Grid)
IF diNrOfEM_OUT_Grid > 0 AND fbNumberDeviceGrid.bNumberIsCalculatet THEN
	Lynus_Standards.GVL_Energy.stDataElectricMeters[diNrOfEM_OUT_Grid].bEnabled := fbEMGrid.stDataEMOutPower.bEnabled;
		Lynus_Standards.GVL_Energy.stDataElectricMeters[diNrOfEM_OUT_Grid].byErrorWarning := fbEMGrid.stDataEMOutPower.byErrorWarning;
			Lynus_Standards.GVL_Energy.stDataElectricMeters[diNrOfEM_OUT_Grid].lrCounterEnergyT1_Consumption := fbEMGrid.stDataEMOutCounter.lrCounterEnergyT1_Consumption;
				Lynus_Standards.GVL_Energy.stDataElectricMeters[diNrOfEM_OUT_Grid].lrCounterEnergyT1_Production := fbEMGrid.stDataEMOutCounter.lrCounterEnergyT1_Production;
					Lynus_Standards.GVL_Energy.stDataElectricMeters[diNrOfEM_OUT_Grid].lrCounterEnergyT2_Consumption := fbEMGrid.stDataEMOutCounter.lrCounterEnergyT2_Consumption;
						Lynus_Standards.GVL_Energy.stDataElectricMeters[diNrOfEM_OUT_Grid].lrCounterEnergyT2_Production := fbEMGrid.stDataEMOutCounter.lrCounterEnergyT2_Production;		
							Lynus_Standards.GVL_Energy.stDataElectricMeters[diNrOfEM_OUT_Grid].lrPower := fbEMGrid.stDataEMOutPower.lrPowerTotal;
								Lynus_Standards.GVL_Energy.stDataElectricMeters[diNrOfEM_OUT_Grid].lrPowerConsumption := fbEMGrid.stDataEMOutPower.lrPowerConsumption;
									Lynus_Standards.GVL_Energy.stDataElectricMeters[diNrOfEM_OUT_Grid].lrPowerProduction := fbEMGrid.stDataEMOutPower.lrPowerProduction;
										Lynus_Standards.GVL_Energy.stDataElectricMeters[diNrOfEM_OUT_Grid].lrTotalCounterEnergy_Consumption := fbEMGrid.stDataEMOutCounter.lrTotalCounterEnergy_Consumption;
											Lynus_Standards.GVL_Energy.stDataElectricMeters[diNrOfEM_OUT_Grid].lrTotalCounterEnergy_Production := fbEMGrid.stDataEMOutCounter.lrTotalCounterEnergy_Production;
END_IF

(*----------------------------------------------------------Save persistent data----------------------------------------------------------------*)

arrPD[1](lrValue:= BOOL_TO_LREAL(bEnable), bEventBasedActive=> );
arrPD[2](lrValue:= BOOL_TO_LREAL(bActivateControl), bEventBasedActive=> );
arrPD[3](lrValue:= BYTE_TO_LREAL(byUnitID), bEventBasedActive=> );
arrPD[4](lrValue:= BYTE_TO_LREAL(byPriority), bEventBasedActive=> );
arrPD[5](lrValue:= DINT_TO_LREAL(diNrOfEMS_IN), bEventBasedActive=> );
arrPD[6](lrValue:= lrMaxCapacityBattery, bEventBasedActive=> );
arrPD[7](lrValue:= DINT_TO_LREAL(diNrOfEMS_IN_CP), bEventBasedActive=> );
PD_String(sText:= sIPAdress, bEventBasedActive=> );

END_FUNCTION_BLOCK

// ---- POUs/prgComEffIO.TcPOU
PROGRAM prgComEffIO
VAR
	fbCom		: FB_MqttCommunicator_V3;
END_VAR

fbCom(
	bConnect				:= TRUE,
	strAuthKey				:=  'BMS99299754422' ,  
	sUserName				:= '32673a79-600a-4644-a67c-4e88e91f75b0', 
	sUserPassword			:= '0be74963-42a9-4df9-8959-e5c2a6d2dc47', 
	time_HeartBeat_sec 		:= T#15S,
	eSavePositionCertificate:= eSavePositionOnPLC.ePostionHardDisk, 
	bConnected=> , 
	bError=> , 
	hrErrorCode=> , 
	eConnectionState=> , 
	eErrorMessage_Out=> );

END_PROGRAM

// ---- POUs/prgPV_2.TcPOU
PROGRAM prgPV_2
VAR
//	fbPVFronius1			: FB_Symo_PV_Inverter_int_1_DM_1_Inverter;
	fbPVFronius1			: FB_Symo_PV_Inverter_INT_1_DM_1_InclDisable;
	fbPVFronius2			: FB_Symo_PV_Inverter_INT_1_DM_1_InclDisable;
	fbPVFronius3			: FB_Symo_PV_Inverter_INT_1_DM_1_InclDisable;
	fbPVFronius4			: FB_Symo_PV_Inverter_FLOAT_1_DM_30_InclDisable;
	fbPVFronius6			: FB_Symo_PV_Inverter_INT_1_DM_1_InclDisable;
	fbPVFronius7			: FB_Symo_PV_Inverter_INT_1_DM_1_InclDisable;
	fbPVInt					: FB_PV_Power;
	fbPVCounter				: FB_EnergyCounter;
	
	lrPowerPV				: LREAL;				//{#lynus.ag#()}
	byErrorWarningPV		: BYTE;					//{#lynus.ag#()}
	
	// extend or reduce amount of PV Inverters
	lrPowerPV_1				: LREAL;				//{#lynus.ag#()}
	lrPowerPV_2				: LREAL;				//{#lynus.ag#()}
	lrPowerPV_3				: LREAL;				//{#lynus.ag#()}
	lrPowerPV_4				: LREAL;				//{#lynus.ag#()}
	lrPowerPV_5				: LREAL;				//{#lynus.ag#()}
	lrPowerPV_6				: LREAL;				//{#lynus.ag#()}
	lrPowerPV_7				: LREAL;				//{#lynus.ag#()}
	m_EnableWrite1: BOOL;
	m_EnableWrite2: BOOL;
	m_EnableWrite3: BOOL;
	m_EnableWrite4: BOOL;
	m_EnableWrite5: BOOL;
	m_EnableWrite6: BOOL;
	m_EnableWrite7: BOOL;
	ton_FeedbackDelay1: Ton;
	ton_FeedbackDelay2: Ton;
	ton_FeedbackDelay3: Ton;
	ton_FeedbackDelay4: Ton;
	ton_FeedbackDelay5: Ton;
	ton_FeedbackDelay6: Ton;
	ton_FeedbackDelay7: Ton;
	tof_FeedbackDelay1: Tof;
	tof_FeedbackDelay2: Tof;
	tof_FeedbackDelay3: Tof;
	tof_FeedbackDelay4: Tof;
	tof_FeedbackDelay5: Tof;
	tof_FeedbackDelay6: Tof;	
	tof_FeedbackDelay7: Tof;	
	
	m_Disable_Inverter1: BOOL;						//{#lynus.ag#()}
	m_Disable_Inverter2: BOOL;						//{#lynus.ag#()}
	m_Disable_Inverter3: BOOL;						//{#lynus.ag#()}
	m_Disable_Inverter4: BOOL;						//{#lynus.ag#()}
	m_Disable_Inverter5: BOOL;						//{#lynus.ag#()}
	m_Disable_Inverter6: BOOL;						//{#lynus.ag#()}
	m_Disable_Inverter7: BOOL;						//{#lynus.ag#()}
	int_SetPointInverter	:INT;					//{#lynus.ag#()}
	m_Enable_ChargingBattery: BOOL;					//{#lynus.ag#()}
	FB_PID_InverterIsland :FB_PID_T;
	FB_Ramp :fb_ramp;
	lrErrorPIDCorrection :LREAL;
	RS_DisableInverte1: Rs;
	RS_DisableInverte2: Rs;
	RS_DisableInverte3: Rs;
	RS_DisableInverte4: Rs;
	RS_DisableInverte5: Rs;
	RS_DisableInverte6: Rs;
	RS_DisableInverte7: Rs;
	int_ControllerType: INT;
	x:REAL;
	m_DisableInverter: BOOL:=FALSE;
	
	lrPV1_Frequency				: LREAL;				//{#lynus.ag#()}
	lrPV1_Frequency10			: LREAL;				//{#lynus.ag#()}
	lrPV1_VoltageL1N			: LREAL;				//{#lynus.ag#()}
	lrPV1_VoltageL2N			: LREAL;				//{#lynus.ag#()}
	lrPV1_VoltageL3N			: LREAL;				//{#lynus.ag#()}
	lrPV1_VoltageL12			: LREAL;				//{#lynus.ag#()}
	lrPV1_VoltageL23			: LREAL;				//{#lynus.ag#()}
	lrPV1_VoltageL31			: LREAL;				//{#lynus.ag#()}
	lrPV2_Frequency				: LREAL;				//{#lynus.ag#()}
	
	m_PVLoadRegluationactive: BOOL;						//{#lynus.ag#()}
	dword_SOC_RegluateStart: DWORD:=85;
	dword_SOC_RegluateStop: DWORD:=90;
	k: INT;
	d: INT;
	lrErrorPIDCorrection_Island: LREAL;

	fb_readOut : FB_ModBus_100Registers_FC3;	
	fb_readOut2 : FB_ModBus_100Registers_FC3;	

	Str_Ip: STRING(20);
	w_Adress:WORD;
	usint_Quantity:USINT;
	arrBuffer_FC3				: ARRAY[1..7,1..6] OF WORD;							


	ton_FrequencyStabilisation: Ton;
	real_Setpoint_PID_In: REAL;					//{#lynus.ag#()}
	int_State_PV1: INT;							//{#lynus.ag#()}
	int_State_PV2: INT;							//{#lynus.ag#()}
	int_State_PV3: INT;							//{#lynus.ag#()}
	int_State_PV4: INT;							//{#lynus.ag#()}
	int_State_PV5: INT;							//{#lynus.ag#()}
	int_State_PV6: INT;							//{#lynus.ag#()}
	int_State_PV7: INT;							//{#lynus.ag#()}
	int_readOut: INT;
	ton_wait_read_out: Ton;
	y: INT;
	z: INT;
	int_Data_Received_old: INT;
	int_SP_ReadOut_PV1: INT;							//{#lynus.ag#()}
	int_SP_ReadOut_PV2: INT;							//{#lynus.ag#()}
	int_SP_ReadOut_PV3: INT;							//{#lynus.ag#()}
	int_SP_ReadOut_PV6: INT;							//{#lynus.ag#()}
	int_SP_ReadOut_PV7: INT;							//{#lynus.ag#()}

	int_SetPointInverter_array:ARRAY[1..7] OF INT;
	FB_Linear_Frequency: FB_LinearEquation;
	lr_ValidFrequency: LREAL;

	real_FrequencyLimit: REAL;						//{#lynus.ag#()}
	

END_VAR
VAR PERSISTENT
	lrCounterPV				: LREAL;				//{#lynus.ag#()}
END_VAR



int_SetPointInverter_array[1] := int_SetPointInverter;
int_SetPointInverter_array[2] := int_SetPointInverter;
int_SetPointInverter_array[3] := int_SetPointInverter;
int_SetPointInverter_array[4] := int_SetPointInverter;
int_SetPointInverter_array[5] := int_SetPointInverter;
int_SetPointInverter_array[6] := int_SetPointInverter;
int_SetPointInverter_array[7] := int_SetPointInverter;
int_SetPointInverter_array[7] := int_SetPointInverter;


//1             Tauro 100            192.168.10.100                 00:03:AC:41:C7:C9
fbPVFronius1(
	bEnable				:= TRUE, 
	sIPAdress			:= '192.168.10.100', 			// modify IP Adress
	b_enableWrite		:= m_EnableWrite1,
	m_DisableInverter	:= m_Disable_Inverter1,
	int_InverterSetpoint:= int_SetPointInverter_array[1],
	stDataSymo10		=> ,
	stDataEMPower_PV	=> , 
	stDataEMCounter_PV	=> , 
	diNrOfEM_OUT_PV		=> );


//2             Tauro 100            192.168.10.101                 00:03:AC:41:C7:DA
fbPVFronius2(
	bEnable				:= TRUE, 
	sIPAdress			:= '192.168.10.101', 			// modify IP Adress
	b_enableWrite		:= m_EnableWrite2,
	m_DisableInverter	:= m_Disable_Inverter2,
	int_InverterSetpoint:= int_SetPointInverter_array[2],
	stDataSymo10		=> ,
	stDataEMPower_PV	=> , 
	stDataEMCounter_PV	=> , 
	diNrOfEM_OUT_PV		=> );

//3             Tauro 50              192.168.10.102                 00:03:AC:42:53:2F	
	fbPVFronius3(
	bEnable				:= TRUE, 
	sIPAdress			:= '192.168.10.102', 			// modify IP Adress
	b_enableWrite		:= m_EnableWrite3,
	m_DisableInverter	:= m_Disable_Inverter3,
	int_InverterSetpoint:= int_SetPointInverter_array[3],
	stDataSymo10		=> ,
	stDataEMPower_PV	=> , 
	stDataEMCounter_PV	=> , 
	diNrOfEM_OUT_PV		=> );

//4             2xSymo27           192.168.10.103                 00:03:AC:32:9F:DC           Node1 und Node2
fbPVFronius4(
	bEnable				:= TRUE, 
	sIPAdress			:= '192.168.10.103', 			// modify IP Adress
	arrUnitID_Inverter	:= ,
	arr_b_EnableWrite	:= ,
	arr_m_DisableInverter := ,
	arrDataSymo10		=> ,
	stDataEMPower_PV	=> , 
	stDataEMCounter_PV	=> , 
	diNrOfEM_OUT_PV		=> );
	
fbPVFronius4.arrUnitID_Inverter[1]:=1;
fbPVFronius4.arrUnitID_Inverter[2]:=2;
fbPVFronius4.arr_b_EnableWrite[1] := m_EnableWrite4;
fbPVFronius4.arr_b_EnableWrite[2] := m_EnableWrite5;
fbPVFronius4.arr_m_DisableInverter[1] := m_Disable_Inverter4;
fbPVFronius4.arr_m_DisableInverter[2] := m_Disable_Inverter5;	
fbPVFronius4.arr_int_InverterSetpoint[1] := int_SetPointInverter_array[4];
fbPVFronius4.arr_int_InverterSetpoint[2] := int_SetPointInverter_array[5];	

//6             Tauro 100            192.168.10.104                 
fbPVFronius6(
	bEnable				:= TRUE, 
	sIPAdress			:= '192.168.10.104', 			// modify IP Adress
	b_enableWrite		:= m_EnableWrite6,
	m_DisableInverter	:= m_Disable_Inverter6,
	int_InverterSetpoint:= int_SetPointInverter_array[6],
	stDataSymo10		=> ,
	stDataEMPower_PV	=> , 
	stDataEMCounter_PV	=> , 
	diNrOfEM_OUT_PV		=> );

//7             Tauro 100            192.168.10.105                 
fbPVFronius7(
	bEnable				:= TRUE, 
	sIPAdress			:= '192.168.10.105', 			// modify IP Adress
	b_enableWrite		:= m_EnableWrite7,
	m_DisableInverter	:= m_Disable_Inverter7,
	int_InverterSetpoint:= int_SetPointInverter_array[7],
	stDataSymo10		=> ,
	stDataEMPower_PV	=> , 
	stDataEMCounter_PV	=> , 
	diNrOfEM_OUT_PV		=> );
	
// extend or reduce amount of PV Inverters
lrPowerPV_1 := fbPVFronius1.stDataEMPower_PV.lrPowerTotal;
lrPowerPV_2 := fbPVFronius2.stDataEMPower_PV.lrPowerTotal;
lrPowerPV_3 := fbPVFronius3.stDataEMPower_PV.lrPowerTotal;

lrPowerPV_4 := fbPVFronius4.arrDataSymo10[1].lrPowerAcInverter;
lrPowerPV_5 := fbPVFronius4.arrDataSymo10[2].lrPowerAcInverter;
lrPowerPV_6 := fbPVFronius6.stDataEMPower_PV.lrPowerTotal;
lrPowerPV_7 := fbPVFronius7.stDataEMPower_PV.lrPowerTotal;

	
fbPVInt(
	bEnable:= TRUE, 
	bPowerDataInvers:= , 
	diNrOfEM_IN_PV:= fbPVFronius1.diNrOfEM_OUT_PV, 
	stDataPv=> , 
	diNrOfPv_OUT=> );
	
//lrPowerPV := fbPVInt.stDataPv.lrPower;
	
lrPowerPV := lrPowerPV_1 + lrPowerPV_2 + lrPowerPV_3 + lrPowerPV_4 + lrPowerPV_5 + lrPowerPV_6 + lrPowerPV_7;
	byErrorWarningPV := fbPVInt.stDataPv.byErrorWarning;

// EnergyCounter
fbPVCounter(
	byActiveTariff:= 1, 
	lrPowerInput:= 0 - lrPowerPV, 
	lrTotalCounterEnergy_Consumption=> , 
	lrTotalCounterEnergy_Production=> , 
	lrCounterEnergyT1_Consumption=> , 
	lrCounterEnergyT2_Consumption=> , 
	lrCounterEnergyT1_Production=> , 
	lrCounterEnergyT2_Production=> );
	
IF fbPVCounter.lrTotalCounterEnergy_Production > lrCounterPV THEN  	
	lrCounterPV := fbPVCounter.lrTotalCounterEnergy_Production;
END_IF




// only done for disabling the solar inverter in case negative mains power / back feeding

IF (*prgGrid.lrPowerGrid < -1*) prgBattery.dwSOCBattery>95 THEN
	ton_FeedbackDelay1.In := TRUE;		// start timer for feeding back delay. 
	ton_FeedbackDelay2.In := TRUE;		// start timer for feeding back delay. 
	ton_FeedbackDelay3.In := TRUE;		// start timer for feeding back delay. 
	ton_FeedbackDelay4.In := TRUE;		// start timer for feeding back delay. 
	ton_FeedbackDelay5.In := TRUE;		// start timer for feeding back delay. 
	ton_FeedbackDelay6.In := TRUE;		// start timer for feeding back delay. 
	ton_FeedbackDelay7.In := TRUE;		// start timer for feeding back delay. 

	tof_FeedbackDelay1.IN :=TRUE;
	tof_FeedbackDelay2.IN :=TRUE;
	tof_FeedbackDelay3.IN :=TRUE;
	tof_FeedbackDelay4.IN :=TRUE;
	tof_FeedbackDelay5.IN :=TRUE;
	tof_FeedbackDelay6.IN :=TRUE;
	tof_FeedbackDelay7.IN :=TRUE;
ELSIF (*prgGrid.lrPowerGrid > 1*) prgBattery.dwSOCBattery<90 THEN
	ton_FeedbackDelay1.In := FALSE;		// start timer for feeding back delay. 
	ton_FeedbackDelay2.In := FALSE;		// start timer for feeding back delay. 
	ton_FeedbackDelay3.In := FALSE;		// start timer for feeding back delay. 
	ton_FeedbackDelay4.In := FALSE;		// start timer for feeding back delay. 
	ton_FeedbackDelay5.In := FALSE;		// start timer for feeding back delay. 
	ton_FeedbackDelay6.In := FALSE;		// start timer for feeding back delay. 
	ton_FeedbackDelay7.In := FALSE;		// start timer for feeding back delay. 

	IF (*prgGrid.fbGrid.fbGrid.stDataGridOut.lrPower > 5*) prgBattery.dwSOCBattery<90 THEN 
		tof_FeedbackDelay1.IN :=FALSE;
	END_IF
	IF (*prgGrid.fbGrid.fbGrid.stDataGridOut.lrPower > 5*) prgBattery.dwSOCBattery<88 THEN 
		tof_FeedbackDelay2.IN :=FALSE;
	END_IF
	tof_FeedbackDelay3.IN :=FALSE;
	tof_FeedbackDelay4.IN :=FALSE;
	tof_FeedbackDelay5.IN :=FALSE;
	tof_FeedbackDelay6.IN :=FALSE;
	tof_FeedbackDelay7.IN :=FALSE;	
END_IF
ton_FeedbackDelay1 ( PT:= T#30S,Q => );		// switch of  inverters1 if feeding back
ton_FeedbackDelay2 ( PT:= T#60S,Q => );		// switch of  inverters2 if feeding back
ton_FeedbackDelay3 ( PT:= T#90S,Q => );		// switch of  inverters3 if feeding back
ton_FeedbackDelay4 ( PT:= T#120S,Q => );		// switch of  inverters4 if feeding back
ton_FeedbackDelay5 ( PT:= T#150S,Q => );		// switch of  inverters5 if feeding back
ton_FeedbackDelay6 ( PT:= T#170S,Q => );		// switch of  inverters6 if feeding back
ton_FeedbackDelay7 ( PT:= T#190S,Q => );		// switch of  inverters7 if feeding back

tof_FeedbackDelay1 ( PT:= T#30S,Q => );		// switch on delay inverters1 
tof_FeedbackDelay2 ( PT:= T#60S,Q => );		// switch on delay inverters2 
tof_FeedbackDelay3 ( PT:= T#90S,Q => );		// switch on delay inverters3 
tof_FeedbackDelay4 ( PT:= T#120S,Q => );		// switch on delay inverters4 
tof_FeedbackDelay5 ( PT:= T#150S,Q => );		// switch on delay inverters5 
tof_FeedbackDelay6 ( PT:= T#170S,Q => );		// switch on delay inverters6 
tof_FeedbackDelay7 ( PT:= T#190S,Q => );		// switch on delay inverters7 

RS_DisableInverte1 (Set := ton_FeedbackDelay1.Q OR prgGrid.lrPowerGrid < -50 OR m_DisableInverter, Reset1 := NOT tof_FeedbackDelay1.Q AND NOT m_DisableInverter, Q1 => m_Disable_Inverter1);
RS_DisableInverte2 (Set := ton_FeedbackDelay2.Q OR prgGrid.lrPowerGrid < -50 OR m_DisableInverter, Reset1 := NOT tof_FeedbackDelay2.Q AND NOT m_DisableInverter, Q1 => m_Disable_Inverter2);
RS_DisableInverte3 (Set := ton_FeedbackDelay3.Q OR prgGrid.lrPowerGrid < -50 OR m_DisableInverter, Reset1 := NOT tof_FeedbackDelay3.Q AND NOT m_DisableInverter, Q1 => m_Disable_Inverter3);
RS_DisableInverte4 (Set := ton_FeedbackDelay4.Q OR prgGrid.lrPowerGrid < -50 OR m_DisableInverter, Reset1 := NOT tof_FeedbackDelay4.Q AND NOT m_DisableInverter, Q1 => m_Disable_Inverter4);
RS_DisableInverte5 (Set := ton_FeedbackDelay5.Q OR prgGrid.lrPowerGrid < -50 OR m_DisableInverter, Reset1 := NOT tof_FeedbackDelay5.Q AND NOT m_DisableInverter, Q1 => m_Disable_Inverter5);
RS_DisableInverte6 (Set := ton_FeedbackDelay6.Q OR prgGrid.lrPowerGrid < -50 OR m_DisableInverter, Reset1 := NOT tof_FeedbackDelay6.Q AND NOT m_DisableInverter, Q1 => m_Disable_Inverter6);
RS_DisableInverte7 (Set := ton_FeedbackDelay7.Q OR prgGrid.lrPowerGrid < -50 OR m_DisableInverter, Reset1 := NOT tof_FeedbackDelay7.Q AND NOT m_DisableInverter, Q1 => m_Disable_Inverter7);

IF m_DisableInverter THEN
	m_Disable_Inverter1:=TRUE;
	m_Disable_Inverter2:=TRUE;
	m_Disable_Inverter3:=TRUE;
	m_Disable_Inverter4:=TRUE;
	m_Disable_Inverter5:=TRUE;
	m_Disable_Inverter6:=TRUE;
	m_Disable_Inverter7:=TRUE;
END_IF
	

// enable write function to all inverters
m_EnableWrite1:=TRUE;
m_EnableWrite2:=TRUE;
m_EnableWrite3:=TRUE;
m_EnableWrite4:=TRUE;
m_EnableWrite5:=TRUE;
m_EnableWrite6:=TRUE;
m_EnableWrite7:=TRUE;


// calculate setpoint for PV Island operation
IF prgBattery.dwSOCBattery< dword_SOC_RegluateStart AND prgBattery.fbBattery.stDataXelectrix.eGridState = 2 THEN
	// is in Island operation and SOC below 89 % then let the PV make max power 
(*	FB_PID_InverterIsland.bEnable := FALSE;
	int_SetPointInverter := 10000;
	m_PVLoadRegluationactive := FALSE;
	m_DisableInverter := FALSE;
*)
	
	FB_PID_InverterIsland.bEnable := TRUE;
	FB_PID_InverterIsland.rSetpoint := lreal_to_real(45+ (prgHouse.lrPowerHouse)/5);
	FB_PID_InverterIsland.rSetpoint := LIMIT(0,FB_PID_InverterIsland.rSetpoint,100);
	int_SetPointInverter := REAL_TO_INT(FB_PID_InverterIsland.rQController);
	m_PVLoadRegluationactive := TRUE;
	m_DisableInverter := FALSE;
	// limit setpoint if frequency is high
	IF lrPV1_Frequency>=50.2 AND lrPV1_Frequency<50.4 THEN
		int_SetPointInverter := 8000;
	ELSIF lrPV1_Frequency>=50.4 AND lrPV1_Frequency<50.8 THEN
		int_SetPointInverter := 5000;
	ELSIF lrPV1_Frequency>=50.8 AND lrPV1_Frequency<51.0 THEN
		int_SetPointInverter := 2500;
	ELSIF lrPV1_Frequency>=51 THEN
		int_SetPointInverter := 1000;
	END_IF	
	FB_PID_InverterIsland.rMaxValue := 10000;
ELSIF prgBattery.dwSOCBattery> dword_SOC_RegluateStop+2 AND prgBattery.fbBattery.stDataXelectrix.eGridState = 2 THEN // "+2" for adding a hysteresis befor shutting down the pv inverters
	// is in Island operation and SOC above max SOC +2  
	FB_PID_InverterIsland.bEnable := FALSE;
	int_SetPointInverter := 0;
	m_PVLoadRegluationactive := FALSE;
	m_DisableInverter := TRUE;
	FB_PID_InverterIsland.rMaxValue := 10000;
ELSIF prgBattery.dwSOCBattery>= dword_SOC_RegluateStop AND prgBattery.dwSOCBattery< dword_SOC_RegluateStop+ 1 AND prgBattery.fbBattery.stDataXelectrix.eGridState = 2 THEN 
	// is in Island operation and SOC above max SOC  --> PV Setpoint = house power 
	FB_PID_InverterIsland.bEnable := TRUE;
	FB_PID_InverterIsland.rSetpoint := LREAL_TO_REAL(prgHouse.lrPowerHouse)/5;
	FB_PID_InverterIsland.rSetpoint := LIMIT(0,FB_PID_InverterIsland.rSetpoint,100);
	int_SetPointInverter := REAL_TO_INT(FB_PID_InverterIsland.rQController);
	m_PVLoadRegluationactive := TRUE;
	m_DisableInverter := FALSE;
	FB_PID_InverterIsland.rMaxValue := 10000;
ELSIF prgBattery.fbBattery.stDataXelectrix.eGridState = 2 THEN
	FB_PID_InverterIsland.bEnable := TRUE;
	m_DisableInverter := FALSE;
	m_PVLoadRegluationactive := TRUE;
	(*IF dword_SOC_RegluateStart>0 AND dword_SOC_RegluateStop>0 AND dword_SOC_RegluateStop<>dword_SOC_RegluateStart THEN // calculate k & d for y = k*x+d;
					// dword_SOC_RegluateStart   --> 100% inverter power
					// dword_SOC_RegluateStop    --> 0% inverter power
		k := (100-0)/(DWORD_TO_INT(dword_SOC_RegluateStart) - DWORD_TO_INT(dword_SOC_RegluateStop));
		d := -(k*DWORD_TO_INT(dword_SOC_RegluateStop));
	END_IF
	
	FB_PID_InverterIsland.rSetpoint := k* DWORD_TO_REAL(prgBattery.dwSOCBattery) + d;
	FB_PID_InverterIsland.rSetpoint := LIMIT(0,FB_PID_InverterIsland.rSetpoint,100);
	*)
	IF dword_SOC_RegluateStart>0 AND dword_SOC_RegluateStop>0 AND dword_SOC_RegluateStop<>dword_SOC_RegluateStart  AND ton_FrequencyStabilisation.Q THEN
		IF prgBattery.dwSOCBattery < dword_SOC_RegluateStart THEN
			FB_PID_InverterIsland.rSetpoint :=LREAL_TO_REAL( 1 + (prgHouse.lrPowerHouse)/5);
		ELSIF prgBattery.dwSOCBattery >= dword_SOC_RegluateStart AND prgBattery.dwSOCBattery <= (dword_SOC_RegluateStop - (dword_SOC_RegluateStop-dword_SOC_RegluateStart)/2) THEN
			FB_PID_InverterIsland.rSetpoint := LREAL_TO_REAL(10 + (prgHouse.lrPowerHouse)/5);
		ELSIF prgBattery.dwSOCBattery > (dword_SOC_RegluateStart+ (dword_SOC_RegluateStop-dword_SOC_RegluateStart)/2) AND prgBattery.dwSOCBattery <= dword_SOC_RegluateStop THEN
			FB_PID_InverterIsland.rSetpoint := LREAL_TO_REAL(4 + (prgHouse.lrPowerHouse)/5);
		ELSE	
			FB_PID_InverterIsland.rSetpoint := LREAL_TO_REAL(15 + (prgHouse.lrPowerHouse)/5);
		END_IF
	END_IF	
	int_SetPointInverter := REAL_TO_INT(FB_PID_InverterIsland.rQController);
		// limit setpoint if frequency is high
	IF lrPV1_Frequency>=50.2 AND lrPV1_Frequency<50.4 THEN
		//int_SetPointInverter := 1000;
		FB_PID_InverterIsland.rMaxValue := 800;
		FB_PID_InverterIsland.rSetpoint := LREAL_TO_REAL(5+(prgHouse.lrPowerHouse)/5);
	ELSIF lrPV1_Frequency>=50.4 AND lrPV1_Frequency<50.8 THEN
		// int_SetPointInverter := 500;
		FB_PID_InverterIsland.rMaxValue := 400;
		FB_PID_InverterIsland.rSetpoint := LREAL_TO_REAL(3+(prgHouse.lrPowerHouse)/5);
	ELSIF lrPV1_Frequency>=50.8 AND lrPV1_Frequency<51.0 THEN
		//int_SetPointInverter := 200;
		FB_PID_InverterIsland.rMaxValue := 200;
		FB_PID_InverterIsland.rSetpoint := LREAL_TO_REAL(2+(prgHouse.lrPowerHouse)/5);
	ELSIF lrPV1_Frequency>=51 THEN
		// int_SetPointInverter := 100;
		FB_PID_InverterIsland.rMaxValue := 100;
		FB_PID_InverterIsland.rSetpoint := LREAL_TO_REAL((prgHouse.lrPowerHouse)/5);
	ELSE
		FB_PID_InverterIsland.rMaxValue := 10000;	
	END_IF	
END_IF

// limit setpoint if frequency is high
// linear Equation Frequency
//find out which invreter PV1 or PV1 has a valid frequency
IF lrPV1_Frequency<> 0 THEN 
	lr_ValidFrequency := lrPV1_Frequency;
ELSIF lrPV2_Frequency<> 0 THEN 
	lr_ValidFrequency := lrPV2_Frequency;
ELSIF fbPVFronius3.stDataEMPower_PV.lrFrequency <> 0 THEN
	lr_ValidFrequency := fbPVFronius3.stDataEMPower_PV.lrFrequency;
ELSIF fbPVFronius6.stDataEMPower_PV.lrFrequency <> 0 THEN
	lr_ValidFrequency := fbPVFronius6.stDataEMPower_PV.lrFrequency;
ELSIF fbPVFronius7.stDataEMPower_PV.lrFrequency <> 0 THEN
	lr_ValidFrequency := fbPVFronius7.stDataEMPower_PV.lrFrequency;
ELSE
	lr_ValidFrequency := 0;
END_IF

FB_Linear_Frequency(
	x1:= 50.1, 
	y1:= 10000, 
	x2:= 51, 
	y2:= 0, 
	x:= LREAL_TO_REAL(lr_ValidFrequency), 
	y=> real_FrequencyLimit );
real_FrequencyLimit := LIMIT(0,real_FrequencyLimit,10000);
FB_PID_InverterIsland.rMaxValue := real_FrequencyLimit;

ton_FrequencyStabilisation(	In := lrPV1_Frequency<=50,
							PT :=T#1M); 


FB_PID_InverterIsland(
	bEnable:= , 
	rSetpoint:= , 
	udiIValue:= , 
	udiDValue:= 0, 
	udiDamping:= 0, 
	rPValue:= , 
	rMaxValue:= , 
	rMinValue:= 100, 
	rNeutralZone:= 1, 
	bDirection:= FALSE, 
	rActualValue:= LREAL_TO_REAL(lrPowerPV)/5,	// 500 kW = 100% 
	rQController=> );
	
lrErrorPIDCorrection_Island := ABS(FB_PID_InverterIsland.rSetpoint - FB_PID_InverterIsland.rActualValue);	
real_Setpoint_PID_In := FB_PID_InverterIsland.rSetpoint;



//Controller weighting
	FB_PID_InverterIsland.rPValue := 2; 
	FB_PID_InverterIsland.udiIValue := 275;
	

// record additinal values
lrPV1_Frequency 	:= fbPVfronius1.stDataEMPower_PV.lrFrequency;
lrPV2_Frequency 	:= fbPVfronius2.stDataEMPower_PV.lrFrequency;
lrPV1_Frequency10	:= fbPVfronius1.stDataEMPower_PV.lrFrequency*10;
lrPV1_VoltageL1N	:= fbPVfronius1.stDataEMPower_PV.lrVoltageL1N;
lrPV1_VoltageL2N	:= fbPVfronius1.stDataEMPower_PV.lrVoltageL2N;
lrPV1_VoltageL3N	:= fbPVfronius1.stDataEMPower_PV.lrVoltageL3N;
lrPV1_VoltageL12	:= fbPVfronius1.stDataEMPower_PV.lrVoltageL1L2;
lrPV1_VoltageL23	:= fbPVfronius1.stDataEMPower_PV.lrVoltageL2L3;
lrPV1_VoltageL31	:= fbPVfronius1.stDataEMPower_PV.lrVoltageL3L1;


	
int_State_PV1 := prgPV.fbPVFronius1.stDataSymo10.eOperatingStateInverter;
int_State_PV2 := prgPV.fbPVFronius2.stDataSymo10.eOperatingStateInverter;
int_State_PV3 := prgPV.fbPVFronius3.stDataSymo10.eOperatingStateInverter;
int_State_PV4 := prgPV.fbPVFronius4.arrDataSymo10[1].eOperatingStateInverter;
int_State_PV5 := prgPV.fbPVFronius4.arrDataSymo10[2].eOperatingStateInverter;
int_State_PV6 := prgPV.fbPVFronius6.stDataSymo10.eOperatingStateInverter;
int_State_PV7 := prgPV.fbPVFronius7.stDataSymo10.eOperatingStateInverter;




// read out setpoints
CASE int_readOut OF
	0: // wait state
		fb_readOut.m_Enable := FALSE;
		ton_wait_read_out.IN := TRUE;
		IF ton_wait_read_out.Q THEN
			ton_wait_read_out.IN := FALSE;
			int_readOut := int_readOut +1;
		END_IF
	1: // read out IP 192.168.10.100 PV1 
		fb_readOut.m_Enable := TRUE;
		Str_Ip := '192.168.10.100';
		usint_Quantity := 6;
		w_Adress := 40231;
		int_readOut := int_readOut +1;
	2: // wait for received values	
		ton_wait_read_out.IN := TRUE;
		IF NOT fb_readOut.fbMBRead_FC3.bBusy AND int_Data_Received_old <> fb_readout.int_Data_Received  THEN
			y:=1;
			FOR z:=1 TO 6 BY 1 DO
				arrBuffer_FC3[y,z] := fb_readOut.w_Array_Received[z];
			END_FOR
			fb_readOut.m_Enable := FALSE;
			ton_wait_read_out.IN := FALSE;
			int_readOut := int_readOut +1;	
		ELSIF fb_readOut.fbMBRead_FC3.bError THEN
			fb_readOut.m_Enable := FALSE;
			ton_wait_read_out.IN := FALSE;
			int_readOut := int_readOut +1;		
		ELSIF ton_wait_read_out.Q THEN
			fb_readOut.m_Enable := FALSE;
			ton_wait_read_out.IN := FALSE;
			int_readOut := int_readOut +1;		
		END_IF
	3: // wait state
		fb_readOut.m_Enable := FALSE;
		ton_wait_read_out.IN := TRUE;
		IF ton_wait_read_out.Q THEN
			ton_wait_read_out.IN := FALSE;
			int_readOut := int_readOut +1;
		END_IF
	4: // read out IP 192.168.10.101 PV2 
		fb_readOut.m_Enable := TRUE;
		Str_Ip := '192.168.10.101';
		usint_Quantity := 6;
		w_Adress := 40231;
		int_Data_Received_old := fb_readout.int_Data_Received;
		int_readOut := int_readOut +1;
	5: // wait for received values	
		ton_wait_read_out.IN := TRUE;
		IF NOT fb_readOut.fbMBRead_FC3.bBusy AND int_Data_Received_old <> fb_readout.int_Data_Received  THEN
			y:=2;
			FOR z:=1 TO 6 BY 1 DO
				arrBuffer_FC3[y,z] := fb_readOut.w_Array_Received[z];
			END_FOR
			fb_readOut.m_Enable := FALSE;
			ton_wait_read_out.IN := FALSE;
			int_readOut := int_readOut +1;	
		ELSIF fb_readOut.fbMBRead_FC3.bError THEN
			fb_readOut.m_Enable := FALSE;
			ton_wait_read_out.IN := FALSE;
			int_readOut := int_readOut +1;		
		ELSIF ton_wait_read_out.Q THEN
			fb_readOut.m_Enable := FALSE;
			ton_wait_read_out.IN := FALSE;
			int_readOut := int_readOut +1;		
		END_IF
	6: // wait state
		fb_readOut.m_Enable := FALSE;
		ton_wait_read_out.IN := TRUE;
		IF ton_wait_read_out.Q THEN
			ton_wait_read_out.IN := FALSE;
			int_readOut := int_readOut +1;
		END_IF
	7: // read out IP 192.168.10.102 PV3 
		fb_readOut.m_Enable := TRUE;
		Str_Ip := '192.168.10.102';
		usint_Quantity := 6;
		w_Adress := 40231;
		int_readOut := int_readOut +1;
	8: // wait for received values	
		ton_wait_read_out.IN := TRUE;
		IF NOT fb_readOut.fbMBRead_FC3.bBusy AND int_Data_Received_old <> fb_readout.int_Data_Received  THEN
			y:=3;
			FOR z:=1 TO 6 BY 1 DO
				arrBuffer_FC3[y,z] := fb_readOut.w_Array_Received[z];
			END_FOR
			fb_readOut.m_Enable := FALSE;
			ton_wait_read_out.IN := FALSE;
			int_readOut := int_readOut +1;	
		ELSIF fb_readOut.fbMBRead_FC3.bError THEN
			fb_readOut.m_Enable := FALSE;
			ton_wait_read_out.IN := FALSE;
			int_readOut := int_readOut +1;		
		ELSIF ton_wait_read_out.Q THEN
			fb_readOut.m_Enable := FALSE;
			ton_wait_read_out.IN := FALSE;
			int_readOut := int_readOut +1;		
		END_IF
	9: // wait state
		fb_readOut.m_Enable := FALSE;
		ton_wait_read_out.IN := TRUE;
		IF ton_wait_read_out.Q THEN
			ton_wait_read_out.IN := FALSE;
			int_readOut := int_readOut +1;
		END_IF
	10: // read out IP 192.168.10.104 PV6 
		fb_readOut.m_Enable := TRUE;
		Str_Ip := '192.168.10.104';
		usint_Quantity := 6;
		w_Adress := 40231;
		int_Data_Received_old := fb_readout.int_Data_Received;
		int_readOut := int_readOut +1;
	11: // wait for received values	
		ton_wait_read_out.IN := TRUE;
		IF NOT fb_readOut.fbMBRead_FC3.bBusy AND int_Data_Received_old <> fb_readout.int_Data_Received  THEN
			y:=6;
			FOR z:=1 TO 6 BY 1 DO
				arrBuffer_FC3[y,z] := fb_readOut.w_Array_Received[z];
			END_FOR
			fb_readOut.m_Enable := FALSE;
			ton_wait_read_out.IN := FALSE;
			int_readOut := int_readOut +1;	
		ELSIF fb_readOut.fbMBRead_FC3.bError THEN
			fb_readOut.m_Enable := FALSE;
			ton_wait_read_out.IN := FALSE;
			int_readOut := int_readOut +1;		
		ELSIF ton_wait_read_out.Q THEN
			fb_readOut.m_Enable := FALSE;
			ton_wait_read_out.IN := FALSE;
			int_readOut := int_readOut +1;		
		END_IF
	12: // wait state
		fb_readOut.m_Enable := FALSE;
		ton_wait_read_out.IN := TRUE;
		IF ton_wait_read_out.Q THEN
			ton_wait_read_out.IN := FALSE;
			int_readOut := int_readOut +1;
		END_IF
	13: // read out IP 192.168.10.105 PV7 
		fb_readOut.m_Enable := TRUE;
		Str_Ip := '192.168.10.105';
		usint_Quantity := 6;
		w_Adress := 40231;
		int_Data_Received_old := fb_readout.int_Data_Received;
		int_readOut := int_readOut +1;
	14: // wait for received values	
		ton_wait_read_out.IN := TRUE;
		IF NOT fb_readOut.fbMBRead_FC3.bBusy AND int_Data_Received_old <> fb_readout.int_Data_Received  THEN
			y:=7;
			FOR z:=1 TO 6 BY 1 DO
				arrBuffer_FC3[y,z] := fb_readOut.w_Array_Received[z];
			END_FOR
			fb_readOut.m_Enable := FALSE;
			ton_wait_read_out.IN := FALSE;
			int_readOut := int_readOut +1;	
		ELSIF fb_readOut.fbMBRead_FC3.bError THEN
			fb_readOut.m_Enable := FALSE;
			ton_wait_read_out.IN := FALSE;
			int_readOut := int_readOut +1;		
		ELSIF ton_wait_read_out.Q THEN
			fb_readOut.m_Enable := FALSE;
			ton_wait_read_out.IN := FALSE;
			int_readOut := int_readOut +1;		
		END_IF
	15: // read out IP 192.168.10.103 PV3 
		fb_readOut.m_Enable := TRUE;
		Str_Ip := '192.168.10.103';
		usint_Quantity := 6;
		w_Adress := 40241;
		int_Data_Received_old := fb_readout.int_Data_Received;
		int_readOut := int_readOut +1;
	16: // wait for received values	
		ton_wait_read_out.IN := TRUE;
		IF NOT fb_readOut.fbMBRead_FC3.bBusy AND int_Data_Received_old <> fb_readout.int_Data_Received  THEN
			y:=4;
			FOR z:=1 TO 6 BY 1 DO
				arrBuffer_FC3[y,z] := fb_readOut.w_Array_Received[z];
			END_FOR
			fb_readOut.m_Enable := FALSE;
			ton_wait_read_out.IN := FALSE;
			int_readOut := int_readOut +1;	
		ELSIF fb_readOut.fbMBRead_FC3.bError THEN
			fb_readOut.m_Enable := FALSE;
			ton_wait_read_out.IN := FALSE;
			int_readOut := int_readOut +1;		
		ELSIF ton_wait_read_out.Q THEN
			fb_readOut.m_Enable := FALSE;
			ton_wait_read_out.IN := FALSE;
			int_readOut := int_readOut +1;		
		END_IF	
	17:
		int_SP_ReadOut_PV1 := WORD_TO_INT(arrBuffer_FC3[1,2]);
		int_SP_ReadOut_PV2 := WORD_TO_INT(arrBuffer_FC3[2,2]);
		int_SP_ReadOut_PV3 := WORD_TO_INT(arrBuffer_FC3[3,2]);
		int_SP_ReadOut_PV6 := WORD_TO_INT(arrBuffer_FC3[6,2]);
		int_SP_ReadOut_PV7 := WORD_TO_INT(arrBuffer_FC3[7,2]);
		int_readOut := 0;		
END_CASE

ton_wait_read_out( 	In :=,
					PT := T#1S);
					
	
fb_readOut(
	m_Enable:= , 
	str_IPAdress:=Str_Ip , 
	w_Adress:=w_Adress , 
	usint_Quantity:= usint_Quantity, 
	m_PollSuccessful=> , 
	w_Array_Received=> , 
	udint_Error_ID=> );
	
fb_readOut2(
	m_Enable:= , 
	str_IPAdress:= , 
	w_Adress:= , 
	usint_Quantity:= , 
	m_PollSuccessful=> , 
	w_Array_Received=> , 
	udint_Error_ID=> );
fb_readOut2.m_Enable := FALSE;

END_PROGRAM

// ---- POUs/prgPV_3.TcPOU
PROGRAM prgPV_3
VAR
//	fbPVFronius1			: FB_Symo_PV_Inverter_int_1_DM_1_Inverter;
	fbPVFronius1			: FB_Symo_PV_Inverter_INT_1_DM_1_InclDisable;
	fbPVFronius2			: FB_Symo_PV_Inverter_INT_1_DM_1_InclDisable;
	fbPVFronius3			: FB_Symo_PV_Inverter_INT_1_DM_1_InclDisable;
	fbPVFronius4			: FB_Symo_PV_Inverter_FLOAT_1_DM_30_InclDisable;
	fbPVFronius6			: FB_Symo_PV_Inverter_INT_1_DM_1_InclDisable;
	fbPVFronius7			: FB_Symo_PV_Inverter_INT_1_DM_1_InclDisable;
	fbPVInt					: FB_PV_Power;
	fbPVCounter				: FB_EnergyCounter;
	
	lrPowerPV				: LREAL;				//{#lynus.ag#()}
	byErrorWarningPV		: BYTE;					//{#lynus.ag#()}
	
	// extend or reduce amount of PV Inverters
	lrPowerPV_1				: LREAL;				//{#lynus.ag#()}
	lrPowerPV_2				: LREAL;				//{#lynus.ag#()}
	lrPowerPV_3				: LREAL;				//{#lynus.ag#()}
	lrPowerPV_4				: LREAL;				//{#lynus.ag#()}
	lrPowerPV_5				: LREAL;				//{#lynus.ag#()}
	lrPowerPV_6				: LREAL;				//{#lynus.ag#()}
	lrPowerPV_7				: LREAL;				//{#lynus.ag#()}
	m_EnableWrite1: BOOL;
	m_EnableWrite2: BOOL;
	m_EnableWrite3: BOOL;
	m_EnableWrite4: BOOL;
	m_EnableWrite5: BOOL;
	m_EnableWrite6: BOOL;
	m_EnableWrite7: BOOL;
	ton_FeedbackDelay1: Ton;
	ton_FeedbackDelay2: Ton;
	ton_FeedbackDelay3: Ton;
	ton_FeedbackDelay4: Ton;
	ton_FeedbackDelay5: Ton;
	ton_FeedbackDelay6: Ton;
	ton_FeedbackDelay7: Ton;
	tof_FeedbackDelay1: Tof;
	tof_FeedbackDelay2: Tof;
	tof_FeedbackDelay3: Tof;
	tof_FeedbackDelay4: Tof;
	tof_FeedbackDelay5: Tof;
	tof_FeedbackDelay6: Tof;	
	tof_FeedbackDelay7: Tof;	
	
	m_Disable_Inverter1: BOOL;						//{#lynus.ag#()}
	m_Disable_Inverter2: BOOL;						//{#lynus.ag#()}
	m_Disable_Inverter3: BOOL;						//{#lynus.ag#()}
	m_Disable_Inverter4: BOOL;						//{#lynus.ag#()}
	m_Disable_Inverter5: BOOL;						//{#lynus.ag#()}
	m_Disable_Inverter6: BOOL;						//{#lynus.ag#()}
	m_Disable_Inverter7: BOOL;						//{#lynus.ag#()}
	int_SetPointInverter	:INT;					//{#lynus.ag#()}
	m_Enable_ChargingBattery: BOOL;					//{#lynus.ag#()}
	FB_PID_InverterIsland :FB_PID_T;
	FB_Ramp :fb_ramp;
	lrErrorPIDCorrection :LREAL;
	RS_DisableInverte1: Rs;
	RS_DisableInverte2: Rs;
	RS_DisableInverte3: Rs;
	RS_DisableInverte4: Rs;
	RS_DisableInverte5: Rs;
	RS_DisableInverte6: Rs;
	RS_DisableInverte7: Rs;
	int_ControllerType: INT;
	x:REAL;
	m_DisableInverter: BOOL:=FALSE;
	
	lrPV1_Frequency				: LREAL;				//{#lynus.ag#()}
	lrPV1_Frequency10			: LREAL;				//{#lynus.ag#()}
	lrPV1_VoltageL1N			: LREAL;				//{#lynus.ag#()}
	lrPV1_VoltageL2N			: LREAL;				//{#lynus.ag#()}
	lrPV1_VoltageL3N			: LREAL;				//{#lynus.ag#()}
	lrPV1_VoltageL12			: LREAL;				//{#lynus.ag#()}
	lrPV1_VoltageL23			: LREAL;				//{#lynus.ag#()}
	lrPV1_VoltageL31			: LREAL;				//{#lynus.ag#()}
	lrPV2_Frequency				: LREAL;				//{#lynus.ag#()}
	
	m_PVLoadRegluationactive: BOOL;						//{#lynus.ag#()}
	dword_SOC_RegluateStart: DWORD:=85;
	dword_SOC_RegluateStop: DWORD:=90;
	k: INT;
	d: INT;
	lrErrorPIDCorrection_Island: LREAL;

	fb_readOut : FB_ModBus_100Registers_FC3;	
	fb_readOut2 : FB_ModBus_100Registers_FC3;	

	Str_Ip: STRING(20);
	w_Adress:WORD;
	usint_Quantity:USINT;
	arrBuffer_FC3				: ARRAY[1..7,1..6] OF WORD;							


	ton_FrequencyStabilisation: Ton;
	real_Setpoint_PID_In: REAL;					//{#lynus.ag#()}
	int_State_PV1: INT;							//{#lynus.ag#()}
	int_State_PV2: INT;							//{#lynus.ag#()}
	int_State_PV3: INT;							//{#lynus.ag#()}
	int_State_PV4: INT;							//{#lynus.ag#()}
	int_State_PV5: INT;							//{#lynus.ag#()}
	int_State_PV6: INT;							//{#lynus.ag#()}
	int_State_PV7: INT;							//{#lynus.ag#()}
	int_readOut: INT;
	ton_wait_read_out: Ton;
	y: INT;
	z: INT;
	int_Data_Received_old: INT;
	int_SP_ReadOut_PV1: INT;							//{#lynus.ag#()}
	int_SP_ReadOut_PV2: INT;							//{#lynus.ag#()}
	int_SP_ReadOut_PV3: INT;							//{#lynus.ag#()}
	int_SP_ReadOut_PV6: INT;							//{#lynus.ag#()}
	int_SP_ReadOut_PV7: INT;							//{#lynus.ag#()}

	int_SetPointInverter_array:ARRAY[1..7] OF INT;
	FB_Linear_Frequency: FB_LinearEquation;
	lr_ValidFrequency: LREAL;

	real_FrequencyLimit: REAL;						//{#lynus.ag#()}
	
	real_PowerLimit: REAL;
	real_PowerLowerLimit: REAL:=180;
	real_PowerUpperLimit: REAL:=220;
	FB_Linear_SOC: FB_LinearEquation;
	real_SOCLimit: REAL;
	
END_VAR
VAR PERSISTENT
	lrCounterPV				: LREAL;				//{#lynus.ag#()}
END_VAR



int_SetPointInverter_array[1] := int_SetPointInverter;
int_SetPointInverter_array[2] := int_SetPointInverter;
int_SetPointInverter_array[3] := int_SetPointInverter;
int_SetPointInverter_array[4] := int_SetPointInverter;
int_SetPointInverter_array[5] := int_SetPointInverter;
int_SetPointInverter_array[6] := int_SetPointInverter;
int_SetPointInverter_array[7] := int_SetPointInverter;
int_SetPointInverter_array[7] := int_SetPointInverter;


//1             Tauro 100            192.168.10.100                 00:03:AC:41:C7:C9
fbPVFronius1(
	bEnable				:= TRUE, 
	sIPAdress			:= '192.168.10.100', 			// modify IP Adress
	b_enableWrite		:= m_EnableWrite1,
	m_DisableInverter	:= m_Disable_Inverter1,
	int_InverterSetpoint:= int_SetPointInverter_array[1],
	stDataSymo10		=> ,
	stDataEMPower_PV	=> , 
	stDataEMCounter_PV	=> , 
	diNrOfEM_OUT_PV		=> );


//2             Tauro 100            192.168.10.101                 00:03:AC:41:C7:DA
fbPVFronius2(
	bEnable				:= TRUE, 
	sIPAdress			:= '192.168.10.101', 			// modify IP Adress
	b_enableWrite		:= m_EnableWrite2,
	m_DisableInverter	:= m_Disable_Inverter2,
	int_InverterSetpoint:= int_SetPointInverter_array[2],
	stDataSymo10		=> ,
	stDataEMPower_PV	=> , 
	stDataEMCounter_PV	=> , 
	diNrOfEM_OUT_PV		=> );

//3             Tauro 50              192.168.10.102                 00:03:AC:42:53:2F	
	fbPVFronius3(
	bEnable				:= TRUE, 
	sIPAdress			:= '192.168.10.102', 			// modify IP Adress
	b_enableWrite		:= m_EnableWrite3,
	m_DisableInverter	:= m_Disable_Inverter3,
	int_InverterSetpoint:= int_SetPointInverter_array[3],
	stDataSymo10		=> ,
	stDataEMPower_PV	=> , 
	stDataEMCounter_PV	=> , 
	diNrOfEM_OUT_PV		=> );

//4             2xSymo27           192.168.10.103                 00:03:AC:32:9F:DC           Node1 und Node2
fbPVFronius4(
	bEnable				:= TRUE, 
	sIPAdress			:= '192.168.10.103', 			// modify IP Adress
	arrUnitID_Inverter	:= ,
	arr_b_EnableWrite	:= ,
	arr_m_DisableInverter := ,
	arrDataSymo10		=> ,
	stDataEMPower_PV	=> , 
	stDataEMCounter_PV	=> , 
	diNrOfEM_OUT_PV		=> );
	
fbPVFronius4.arrUnitID_Inverter[1]:=1;
fbPVFronius4.arrUnitID_Inverter[2]:=2;
fbPVFronius4.arr_b_EnableWrite[1] := m_EnableWrite4;
fbPVFronius4.arr_b_EnableWrite[2] := m_EnableWrite5;
fbPVFronius4.arr_m_DisableInverter[1] := m_Disable_Inverter4;
fbPVFronius4.arr_m_DisableInverter[2] := m_Disable_Inverter5;	
fbPVFronius4.arr_int_InverterSetpoint[1] := int_SetPointInverter_array[4];
fbPVFronius4.arr_int_InverterSetpoint[2] := int_SetPointInverter_array[5];	

//6             Tauro 100            192.168.10.104                 
fbPVFronius6(
	bEnable				:= TRUE, 
	sIPAdress			:= '192.168.10.104', 			// modify IP Adress
	b_enableWrite		:= m_EnableWrite6,
	m_DisableInverter	:= m_Disable_Inverter6,
	int_InverterSetpoint:= int_SetPointInverter_array[6],
	stDataSymo10		=> ,
	stDataEMPower_PV	=> , 
	stDataEMCounter_PV	=> , 
	diNrOfEM_OUT_PV		=> );

//7             Tauro 100            192.168.10.105                 
fbPVFronius7(
	bEnable				:= TRUE, 
	sIPAdress			:= '192.168.10.105', 			// modify IP Adress
	b_enableWrite		:= m_EnableWrite7,
	m_DisableInverter	:= m_Disable_Inverter7,
	int_InverterSetpoint:= int_SetPointInverter_array[7],
	stDataSymo10		=> ,
	stDataEMPower_PV	=> , 
	stDataEMCounter_PV	=> , 
	diNrOfEM_OUT_PV		=> );
	
// extend or reduce amount of PV Inverters
lrPowerPV_1 := fbPVFronius1.stDataEMPower_PV.lrPowerTotal;
lrPowerPV_2 := fbPVFronius2.stDataEMPower_PV.lrPowerTotal;
lrPowerPV_3 := fbPVFronius3.stDataEMPower_PV.lrPowerTotal;

lrPowerPV_4 := fbPVFronius4.arrDataSymo10[1].lrPowerAcInverter;
lrPowerPV_5 := fbPVFronius4.arrDataSymo10[2].lrPowerAcInverter;
lrPowerPV_6 := fbPVFronius6.stDataEMPower_PV.lrPowerTotal;
lrPowerPV_7 := fbPVFronius7.stDataEMPower_PV.lrPowerTotal;

	
fbPVInt(
	bEnable:= TRUE, 
	bPowerDataInvers:= , 
	diNrOfEM_IN_PV:= fbPVFronius1.diNrOfEM_OUT_PV, 
	stDataPv=> , 
	diNrOfPv_OUT=> );
	
//lrPowerPV := fbPVInt.stDataPv.lrPower;
	
lrPowerPV := lrPowerPV_1 + lrPowerPV_2 + lrPowerPV_3 + lrPowerPV_4 + lrPowerPV_5 + lrPowerPV_6 + lrPowerPV_7;
	byErrorWarningPV := fbPVInt.stDataPv.byErrorWarning;

// EnergyCounter
fbPVCounter(
	byActiveTariff:= 1, 
	lrPowerInput:= 0 - lrPowerPV, 
	lrTotalCounterEnergy_Consumption=> , 
	lrTotalCounterEnergy_Production=> , 
	lrCounterEnergyT1_Consumption=> , 
	lrCounterEnergyT2_Consumption=> , 
	lrCounterEnergyT1_Production=> , 
	lrCounterEnergyT2_Production=> );
	
IF fbPVCounter.lrTotalCounterEnergy_Production > lrCounterPV THEN  	
	lrCounterPV := fbPVCounter.lrTotalCounterEnergy_Production;
END_IF




// only done for disabling the solar inverter in case negative mains power / back feeding

IF (*prgGrid.lrPowerGrid < -1*) prgBattery.dwSOCBattery>95 THEN
	ton_FeedbackDelay1.In := TRUE;		// start timer for feeding back delay. 
	ton_FeedbackDelay2.In := TRUE;		// start timer for feeding back delay. 
	ton_FeedbackDelay3.In := TRUE;		// start timer for feeding back delay. 
	ton_FeedbackDelay4.In := TRUE;		// start timer for feeding back delay. 
	ton_FeedbackDelay5.In := TRUE;		// start timer for feeding back delay. 
	ton_FeedbackDelay6.In := TRUE;		// start timer for feeding back delay. 
	ton_FeedbackDelay7.In := TRUE;		// start timer for feeding back delay. 

	tof_FeedbackDelay1.IN :=TRUE;
	tof_FeedbackDelay2.IN :=TRUE;
	tof_FeedbackDelay3.IN :=TRUE;
	tof_FeedbackDelay4.IN :=TRUE;
	tof_FeedbackDelay5.IN :=TRUE;
	tof_FeedbackDelay6.IN :=TRUE;
	tof_FeedbackDelay7.IN :=TRUE;
ELSIF (*prgGrid.lrPowerGrid > 1*) prgBattery.dwSOCBattery<90 THEN
	ton_FeedbackDelay1.In := FALSE;		// start timer for feeding back delay. 
	ton_FeedbackDelay2.In := FALSE;		// start timer for feeding back delay. 
	ton_FeedbackDelay3.In := FALSE;		// start timer for feeding back delay. 
	ton_FeedbackDelay4.In := FALSE;		// start timer for feeding back delay. 
	ton_FeedbackDelay5.In := FALSE;		// start timer for feeding back delay. 
	ton_FeedbackDelay6.In := FALSE;		// start timer for feeding back delay. 
	ton_FeedbackDelay7.In := FALSE;		// start timer for feeding back delay. 

	IF (*prgGrid.fbGrid.fbGrid.stDataGridOut.lrPower > 5*) prgBattery.dwSOCBattery<90 THEN 
		tof_FeedbackDelay1.IN :=FALSE;
	END_IF
	IF (*prgGrid.fbGrid.fbGrid.stDataGridOut.lrPower > 5*) prgBattery.dwSOCBattery<88 THEN 
		tof_FeedbackDelay2.IN :=FALSE;
	END_IF
	tof_FeedbackDelay3.IN :=FALSE;
	tof_FeedbackDelay4.IN :=FALSE;
	tof_FeedbackDelay5.IN :=FALSE;
	tof_FeedbackDelay6.IN :=FALSE;
	tof_FeedbackDelay7.IN :=FALSE;	
END_IF
ton_FeedbackDelay1 ( PT:= T#30S,Q => );		// switch of  inverters1 if feeding back
ton_FeedbackDelay2 ( PT:= T#60S,Q => );		// switch of  inverters2 if feeding back
ton_FeedbackDelay3 ( PT:= T#90S,Q => );		// switch of  inverters3 if feeding back
ton_FeedbackDelay4 ( PT:= T#120S,Q => );		// switch of  inverters4 if feeding back
ton_FeedbackDelay5 ( PT:= T#150S,Q => );		// switch of  inverters5 if feeding back
ton_FeedbackDelay6 ( PT:= T#170S,Q => );		// switch of  inverters6 if feeding back
ton_FeedbackDelay7 ( PT:= T#190S,Q => );		// switch of  inverters7 if feeding back

tof_FeedbackDelay1 ( PT:= T#30S,Q => );		// switch on delay inverters1 
tof_FeedbackDelay2 ( PT:= T#60S,Q => );		// switch on delay inverters2 
tof_FeedbackDelay3 ( PT:= T#90S,Q => );		// switch on delay inverters3 
tof_FeedbackDelay4 ( PT:= T#120S,Q => );		// switch on delay inverters4 
tof_FeedbackDelay5 ( PT:= T#150S,Q => );		// switch on delay inverters5 
tof_FeedbackDelay6 ( PT:= T#170S,Q => );		// switch on delay inverters6 
tof_FeedbackDelay7 ( PT:= T#190S,Q => );		// switch on delay inverters7 

RS_DisableInverte1 (Set := ton_FeedbackDelay1.Q OR prgGrid.lrPowerGrid < -50 OR m_DisableInverter, Reset1 := NOT tof_FeedbackDelay1.Q AND NOT m_DisableInverter, Q1 => m_Disable_Inverter1);
RS_DisableInverte2 (Set := ton_FeedbackDelay2.Q OR prgGrid.lrPowerGrid < -50 OR m_DisableInverter, Reset1 := NOT tof_FeedbackDelay2.Q AND NOT m_DisableInverter, Q1 => m_Disable_Inverter2);
RS_DisableInverte3 (Set := ton_FeedbackDelay3.Q OR prgGrid.lrPowerGrid < -50 OR m_DisableInverter, Reset1 := NOT tof_FeedbackDelay3.Q AND NOT m_DisableInverter, Q1 => m_Disable_Inverter3);
RS_DisableInverte4 (Set := ton_FeedbackDelay4.Q OR prgGrid.lrPowerGrid < -50 OR m_DisableInverter, Reset1 := NOT tof_FeedbackDelay4.Q AND NOT m_DisableInverter, Q1 => m_Disable_Inverter4);
RS_DisableInverte5 (Set := ton_FeedbackDelay5.Q OR prgGrid.lrPowerGrid < -50 OR m_DisableInverter, Reset1 := NOT tof_FeedbackDelay5.Q AND NOT m_DisableInverter, Q1 => m_Disable_Inverter5);
RS_DisableInverte6 (Set := ton_FeedbackDelay6.Q OR prgGrid.lrPowerGrid < -50 OR m_DisableInverter, Reset1 := NOT tof_FeedbackDelay6.Q AND NOT m_DisableInverter, Q1 => m_Disable_Inverter6);
RS_DisableInverte7 (Set := ton_FeedbackDelay7.Q OR prgGrid.lrPowerGrid < -50 OR m_DisableInverter, Reset1 := NOT tof_FeedbackDelay7.Q AND NOT m_DisableInverter, Q1 => m_Disable_Inverter7);

IF m_DisableInverter THEN
	m_Disable_Inverter1:=TRUE;
	m_Disable_Inverter2:=TRUE;
	m_Disable_Inverter3:=TRUE;
	m_Disable_Inverter4:=TRUE;
	m_Disable_Inverter5:=TRUE;
	m_Disable_Inverter6:=TRUE;
	m_Disable_Inverter7:=TRUE;
ELSE
	m_Disable_Inverter1:=FALSE;
	m_Disable_Inverter2:=FALSE;
	m_Disable_Inverter3:=FALSE;
	m_Disable_Inverter4:=FALSE;
	m_Disable_Inverter5:=FALSE;
	m_Disable_Inverter6:=FALSE;
	m_Disable_Inverter7:=FALSE;
END_IF
	

// enable write function to all inverters
m_EnableWrite1:=TRUE;
m_EnableWrite2:=TRUE;
m_EnableWrite3:=TRUE;
m_EnableWrite4:=TRUE;
m_EnableWrite5:=TRUE;
m_EnableWrite6:=TRUE;
m_EnableWrite7:=TRUE;


// calculate setpoint for PV Island operation
IF prgBattery.fbBattery.stDataXelectrix.eGridState = 2 THEN

	
	FB_PID_InverterIsland.bEnable := TRUE;
	FB_PID_InverterIsland.rSetpoint := (LREAL_TO_REAL((200 *real_SOCLimit)/100+ (prgHouse.lrPowerHouse))/5);
	FB_PID_InverterIsland.rSetpoint := LIMIT(0,FB_PID_InverterIsland.rSetpoint,100);
	int_SetPointInverter := REAL_TO_INT(FB_PID_InverterIsland.rQController);
	m_PVLoadRegluationactive := TRUE;
END_IF

// limit setpoint if frequency is high
// linear Equation Frequency
//find out which invreter PV1 or PV1 has a valid frequency
IF lrPV1_Frequency<> 0 THEN 
	lr_ValidFrequency := lrPV1_Frequency;
ELSIF lrPV2_Frequency<> 0 THEN 
	lr_ValidFrequency := lrPV2_Frequency;
ELSIF fbPVFronius3.stDataEMPower_PV.lrFrequency <> 0 THEN
	lr_ValidFrequency := fbPVFronius3.stDataEMPower_PV.lrFrequency;
ELSIF fbPVFronius6.stDataEMPower_PV.lrFrequency <> 0 THEN
	lr_ValidFrequency := fbPVFronius6.stDataEMPower_PV.lrFrequency;
ELSIF fbPVFronius7.stDataEMPower_PV.lrFrequency <> 0 THEN
	lr_ValidFrequency := fbPVFronius7.stDataEMPower_PV.lrFrequency;
ELSE
	lr_ValidFrequency := 0;
END_IF

FB_Linear_Frequency(
	x1:= 50.1, 
	y1:= 10000, 
	x2:= 50.5, 
	y2:= 0, 
	x:= LREAL_TO_REAL(lr_ValidFrequency), 
	y=> real_FrequencyLimit );
real_FrequencyLimit := LIMIT(0,real_FrequencyLimit,10000);
FB_PID_InverterIsland.rMaxValue := real_FrequencyLimit;

ton_FrequencyStabilisation(	In := lrPV1_Frequency<=50,
							PT :=T#1M); 
// linea Equation SOC

FB_Linear_SOC(
	x1:= DWORD_TO_REAL(dword_SOC_RegluateStart), 
	y1:= 100, 
	x2:= DWORD_TO_REAL(dword_SOC_RegluateStop), 
	y2:= 0, 
	x:= DWORD_TO_REAL(prgBattery.dwSOCBattery), 
	y=> real_SOCLimit);
real_SOCLimit := LIMIT(0,real_SOCLimit,100);


FB_PID_InverterIsland(
	bEnable:= , 
	rSetpoint:= , 
	udiIValue:= , 
	udiDValue:= 0, 
	udiDamping:= 0, 
	rPValue:= , 
	rMaxValue:= , 
	rMinValue:= 100, 
	rNeutralZone:= 1, 
	bDirection:= FALSE, 
	rActualValue:= LREAL_TO_REAL(lrPowerPV)/5,	// 500 kW = 100% 
	rQController=> );
	
lrErrorPIDCorrection_Island := ABS(FB_PID_InverterIsland.rSetpoint - FB_PID_InverterIsland.rActualValue);	
real_Setpoint_PID_In := FB_PID_InverterIsland.rSetpoint;



//Controller weighting
	FB_PID_InverterIsland.rPValue := 2; 
	FB_PID_InverterIsland.udiIValue := 275;
	

// record additinal values
lrPV1_Frequency 	:= fbPVfronius1.stDataEMPower_PV.lrFrequency;
lrPV2_Frequency 	:= fbPVfronius2.stDataEMPower_PV.lrFrequency;
lrPV1_Frequency10	:= fbPVfronius1.stDataEMPower_PV.lrFrequency*10;
lrPV1_VoltageL1N	:= fbPVfronius1.stDataEMPower_PV.lrVoltageL1N;
lrPV1_VoltageL2N	:= fbPVfronius1.stDataEMPower_PV.lrVoltageL2N;
lrPV1_VoltageL3N	:= fbPVfronius1.stDataEMPower_PV.lrVoltageL3N;
lrPV1_VoltageL12	:= fbPVfronius1.stDataEMPower_PV.lrVoltageL1L2;
lrPV1_VoltageL23	:= fbPVfronius1.stDataEMPower_PV.lrVoltageL2L3;
lrPV1_VoltageL31	:= fbPVfronius1.stDataEMPower_PV.lrVoltageL3L1;


	
int_State_PV1 := prgPV.fbPVFronius1.stDataSymo10.eOperatingStateInverter;
int_State_PV2 := prgPV.fbPVFronius2.stDataSymo10.eOperatingStateInverter;
int_State_PV3 := prgPV.fbPVFronius3.stDataSymo10.eOperatingStateInverter;
int_State_PV4 := prgPV.fbPVFronius4.arrDataSymo10[1].eOperatingStateInverter;
int_State_PV5 := prgPV.fbPVFronius4.arrDataSymo10[2].eOperatingStateInverter;
int_State_PV6 := prgPV.fbPVFronius6.stDataSymo10.eOperatingStateInverter;
int_State_PV7 := prgPV.fbPVFronius7.stDataSymo10.eOperatingStateInverter;




